// StandardPLC/Application/SaveEngine/SaveEngineMode_10
PROGRAM SaveEngineMode_10
VAR
(*	DonglitouBlink:BLINK;//0
	DonglitouBlink_biaozhi:BOOL;//0
	DOH_Y50_1: BOOL;//0
	Rotation_late:TOF;//0
	PWM_Y23_SET_Taget: UINT;//0
	PWM_Y24_SET_Taget: UINT;//0
	PWM_Y61_SET_Tatget: UINT;//0
	PWM_Y12_SET_Tatget: UINT;//0
	PWM_Y14_SET_Tatget: UINT;//0
	PWM_Y60_SET_Tatget: UINT;//0
	PWM_Y11_SET_Tatget: UINT;//0
	PWM_Y13_SET_Tatget: UINT;//0
	PWM_Y61_SET_Tatget1: INT;//0
	PWM_Y12_SET_Tatget1: INT;//0
	PWM_Y14_SET_Tatget1: INT;//0
	PWM_Y60_SET_Tatget1: INT;//0
	PWM_Y11_SET_Tatget1: INT;//0
	PWM_Y13_SET_Tatget1: INT;//0
	TIME_200ms:TON;//0
	TIME_400ms:TON;//0
	CANI_JOYX_R_last:UINT;//0
	Sub_Joyx_r: INT;//0
	curve1:curve_quxian;//0
	curve2:curve_quxian;//0
	curve3:curve_quxian;//0
	curve4:curve_quxian;//0
	curve5:curve_quxian;//0
	curve6:curve_quxian;//0
	RAMP1:RAMP_INT;//0
	RAMP2:RAMP_INT;//0
	RAMP3:RAMP_INT;//0
	RAMP4:RAMP_INT;//0
	RAMP5:RAMP_INT;//0
	RAMP6:RAMP_INT;//0
	F_RAMP_1:INT:=250;//0
	PWM_JOYX_R_UP_a:UINT;//0
	PWM_JOYX_R_UP_b:UINT;//0
	
	PWM_JOYX_R_DOWN_a:UINT;//0
	PWM_JOYX_R_DOWN_b:UINT;//0
	
	PWM_JOYY_L_DOWN_a:UINT;//0
	PWM_JOYY_L_DOWN_b:UINT;//0
	
	PWM_JOYY_L_UP_a:UINT;//0
	PWM_JOYY_L_UP_b:UINT;//0
	JOY_PAOTU:BOOL;//0
	TIME_1000_1ms:ton;//0
	tempbool:BOOL;//0
	Rtrig_d1:R_TRIG;//0
	Rtrig_d2:R_TRIG;//0
*)
END_VAR


(*******************节能控制阀主阀主泵输出执行**************************)
	
//ELSIF(GVL_SaveEngine.SaveEngineMode=10)THEN  //下放能量过高模式,先按常规执行
	//GVL_SaveEngine.Y72OutPutState:=0;
	//GVL_SaveEngine.Y71OutPutState:=0;
	GVL_SaveEngine.Y72OutPutState:=0;
	IF Mode10Timer>0 THEN
		GVL_SaveEngine.Y71OutPutState:=0;
	END_IF
	
	DOH_Y56:=FALSE;
	Y73:=FALSE;	
	PWM_Y1_Target:=REAL_TO_UINT(UINT_TO_REAL(PWM_JOYY_L_UP)/1000*(PAR_Y1_PosFull-PAR_Y1_NegFull)+PAR_Y1_NegFull);
	PWM_Y2_Target:=REAL_TO_UINT(UINT_TO_REAL(PWM_JOYY_L_UP)/1000*(PAR_Y2_PosFull-PAR_Y2_NegFull)+PAR_Y2_NegFull);
	PWM_Y8_SET_Target:=REAL_TO_UINT(UINT_TO_REAL(PWM_JOYY_L_UP)/1000*(PAR_Valve1_PosFull-PAR_Valve1_NegFull)+PAR_Valve1_NegFull);
	PWM_Y10_SET_Target:=REAL_TO_UINT(UINT_TO_REAL(PWM_JOYY_L_UP)/1000*(PAR_Valve2_PosFull-PAR_Valve2_NegFull)+PAR_Valve2_NegFull);
	PWM_Y7_SET_Target:=0;
	PWM_Y9_SET_Target:=0;
	PWM_Y33_SET_Target:=370;
	
  //Y33输出处理
	IF PWM_Y33_SET>=PWM_Y33_SET_Target THEN
	PWM_Y33_SET := PWM_Y33_SET_Target;
	END_IF
		
	IF(PWM_Y33_SET<PWM_Y33_SET_Target) THEN
		PWM_Y33_SET:=REAL_TO_UINT(UINT_TO_REAL(PWM_Y33_SET)+JianGE6);
	END_IF
	
	IF DIL_SQ3 THEN
		PWM_Y33_SET:=0;
	END_IF
(*主泵功率控制*)

//区分发动机转速
MainPump_Pressure_Taget1450:=PAR_NegFull_x;
MainPump_Pressure_Taget1600:=PAR_PosFull_x;
MainPump_Pressure_Taget1750:=PAR_Zero_x;
IF EngineSpeedTarget<=1080 THEN SPEED_CASE:=1;
ELSIF EngineSpeedTarget>1080 AND EngineSpeedTarget<=1300 THEN SPEED_CASE:=2;
ELSIF EngineSpeedTarget>1300 AND EngineSpeedTarget<=1520 THEN SPEED_CASE:=3;
ELSIF EngineSpeedTarget>1520 AND EngineSpeedTarget<=1680 THEN SPEED_CASE:=4;
ELSIF EngineSpeedTarget>1680 AND EngineSpeedTarget<=1820 THEN SPEED_CASE:=5;
ELSIF EngineSpeedTarget>1820 THEN SPEED_CASE:=6;;END_IF
//不同转速下的发动机最大功率*)
CASE SPEED_CASE OF
1:  Enginer_Power:=135;
2:  Enginer_Power:=174;
3:  Enginer_Power:=200;
4:  Enginer_Power:=230;
5:  Enginer_Power:=250;
6:  Enginer_Power:=261;
END_CASE
//不同转速下的压力值
IF(CANO_Fubeng_Press>100)THEN
	CASE SPEED_CASE OF
	1:MainPump_Pressure_Taget:=MainPump_Pressure_Taget1000-HELIU_Press_Target1000;
	2:MainPump_Pressure_Taget:=MainPump_Pressure_Taget1200-HELIU_Press_Target1200;
	3:MainPump_Pressure_Taget:=MainPump_Pressure_Taget1450-HELIU_Press_Target1400;
	4:MainPump_Pressure_Taget:=MainPump_Pressure_Taget1600-HELIU_Press_Target1600;
	5:MainPump_Pressure_Taget:=MainPump_Pressure_Taget1750-HELIU_Press_Target1800;
	6:MainPump_Pressure_Taget:=MainPump_Pressure_Taget1900-HELIU_Press_Target1900;
	END_CASE
ELSE
	CASE SPEED_CASE OF
	1:MainPump_Pressure_Taget:=MainPump_Pressure_Taget1000;
	2:MainPump_Pressure_Taget:=MainPump_Pressure_Taget1200;
	3:MainPump_Pressure_Taget:=MainPump_Pressure_Taget1450;
	4:MainPump_Pressure_Taget:=MainPump_Pressure_Taget1600;
	5:MainPump_Pressure_Taget:=MainPump_Pressure_Taget1750;
	6:MainPump_Pressure_Taget:=MainPump_Pressure_Taget1900;
	END_CASE		
END_IF

IF( CANI_ECOSwitch) THEN
	CASE SPEED_CASE OF
	1:MainPump_Pressure_Taget:=MainPump_Pressure_Taget1000-ECO_Press_Target1000;
	2:MainPump_Pressure_Taget:=MainPump_Pressure_Taget1200-ECO_Press_Target1200;
	3:MainPump_Pressure_Taget:=MainPump_Pressure_Taget1450-ECO_Press_Target1400;
	4:MainPump_Pressure_Taget:=MainPump_Pressure_Taget1600-ECO_Press_Target1600;
	5:MainPump_Pressure_Taget:=MainPump_Pressure_Taget1750-ECO_Press_Target1800;
	6:MainPump_Pressure_Taget:=MainPump_Pressure_Taget1900-ECO_Press_Target1900;
	END_CASE
END_IF
MainPump_Pressure:=CANO_MainPUMP_Press1+CANO_MainPUMP_Press2;
//消除滤波
MainPump_Pressure_Subtract:= UINT_TO_INT(MainPump_Pressure-MainPump_Pressure_last1);


//大范围波动
IF MainPump_Pressure_Subtract>270 OR MainPump_Pressure_Subtract<-270 THEN
	Subtract:=TRUE;
ELSE
	Subtract:=FALSE;	
END_IF
	TIME_LvBo4(IN:=Subtract,PT:=T#10MS);
	
IF(TIME_LvBo4.Q) AND (CANO_MainPUMP_Press1>210) THEN 
		MainPump_Pressure_ChangeBool1:=TRUE;
END_IF
	TIME_LvBo1(IN:=MainPump_Pressure_ChangeBool1,PT:=T#2S);
IF(TIME_LvBo1.Q) THEN
	MainPump_Pressure_ChangeBool1 :=FALSE;
END_IF

IF(MainPump_Pressure_ChangeBool1) AND (MainPump_Pressure>MainPump_Pressure_last1) THEN 
	MainPump_Pressure_last1:=MainPump_Pressure;
END_IF

//小范围波动
t_powertime:=TO_TIME(PAR_DeadBand_x);
IF (NOT MainPump_Pressure_ChangeBool1) THEN
	IF(MainPump_Pressure_Subtract>40 OR MainPump_Pressure_Subtract<-40)THEN 
		MainPump_Pressure_ChangeBool:=TRUE;
	ELSE
		MainPump_Pressure_ChangeBool:=FALSE;
	END_IF

	TIME_LvBo2(IN:=MainPump_Pressure_ChangeBool,PT:=t_powertime);
	IF(TIME_LvBo2.Q )THEN
		MainPump_Pressure_last1:=MainPump_Pressure;
	END_IF	
END_IF


IF PowerHead_move AND NOT(MainWinch_move) THEN
		JianGE2:=0.005;
ELSE
	IF(EngineSpeedTarget>1000 AND EngineSpeedTarget<1300)THEN
		JianGE2:=0.005;
	ELSE
		JianGE2:=0.005;
	END_IF
END_IF

IF MainPump_Pressure_last1>MainPump_Pressure_Taget THEN
	Pressure_Coe_Taget:=UINT_TO_REAL(MainPump_Pressure_Taget)/UINT_TO_REAL(MainPump_Pressure_last1);(*压力系数*)
ELSE
	Pressure_Coe_Taget:=1;
END_IF
Pressure_Coe := Pressure_Coe_Taget;


IF MainPump_Pressure_last1>MainPump_Pressure_Taget  THEN
	IF(PWM_Y1_Target>=PAR_Y1_1_NegFull)THEN
		PWM_Y1_Target_OutPut:=REAL_TO_UINT(UINT_TO_REAL(PWM_Y1_Target-PAR_Y1_1_NegFull)*Pressure_Coe+PAR_Y1_1_NegFull);
	END_IF
	IF(PWM_Y2_Target>=PAR_Y1_1_NegFull)THEN
		PWM_Y2_Target_OutPut:=REAL_TO_UINT(UINT_TO_REAL(PWM_Y2_Target-PAR_Y1_1_NegFull)*Pressure_Coe+PAR_Y1_1_NegFull);
	END_IF
ELSE
	PWM_Y1_Target_OutPut:=PWM_Y1_Target;
	PWM_Y2_Target_OutPut:=PWM_Y2_Target;
END_IF

//PWM_Y1_Target_OutPut:=PWM_Y1_Target;
//PWM_Y2_Target_OutPut:=PWM_Y2_Target;


IF(EngineSpeedTarget>CANO_SPEED AND CANO_SPEED>400)THEN
	EngineSpeedSub:=EngineSpeedTarget - CANO_SPEED;
ELSE
	EngineSpeedSub:=0;
END_IF

IF(PWM_Y1_Target_OutPut<300)THEN PWM_Y1_Target_OutPut:=300;END_IF	
IF(PWM_Y2_Target_OutPut<300)THEN PWM_Y2_Target_OutPut:=300;END_IF

RAMP15_IN:=PWM_Y1_Target_OutPut;
RAMP16_IN:=PWM_Y2_Target_OutPut;
(*
RAMP15(
	IN:=UINT_TO_INT(RAMP15_IN), 
	ASCEND:= 300, 
	DESCEND:= 400, 
	TIMEBASE:=T#1000MS , 
	RESET:=FALSE , 
	OUT=>(PWM_Y1_SET));
	
RAMP16(
	IN:=UINT_TO_INT(RAMP16_IN), 
	ASCEND:= 300, 
	DESCEND:= 400, 
	TIMEBASE:=T#1000MS , 
	RESET:=FALSE , 
	OUT=>(PWM_Y2_SET));
	*)
	
	CASE SPEED_CASE OF
                1:F_RAMP_pump:=1500; R_RAMP_pump:=100;                  
                2: 		IF MainWinch_move AND (JiaYa_move OR CANO_JiayaPressure>80)  THEN    //3泵同时起压时，降低主泵的加载速度，避免掉速熄火
                                F_RAMP_pump:=1500; R_RAMP_pump:=100;
                        ELSE
                                F_RAMP_pump:=1500; R_RAMP_pump:=100;//从200降
                                IF  PWM_JOYY_L_UP>10 THEN
                                 F_RAMP_pump:=1500; R_RAMP_pump:=200;
                                END_IF
                        END_IF            
                3:
                        IF MainWinch_move AND (JiaYa_move OR CANO_JiayaPressure>80)  THEN    //3泵同时起压时，降低主泵的加载速度，避免掉速熄火
                                F_RAMP_pump:=1500; R_RAMP_pump:=150;
                        ELSE
                                F_RAMP_pump:=1500; R_RAMP_pump:=TO_INT(PAR_NegFull_y);
                                IF  PWM_JOYY_L_UP>10 THEN
                                 F_RAMP_pump:=1500; R_RAMP_pump:=300;
                                END_IF
                        END_IF                
                4:
                        IF MainWinch_move AND (JiaYa_move OR CANO_JiayaPressure>80)  THEN
                                F_RAMP_pump:=1500; R_RAMP_pump:=150;
                        ELSE
                                F_RAMP_pump:=1500; R_RAMP_pump:=TO_INT(PAR_PosFull_y);//从200降
                                IF  PWM_JOYY_L_UP>10 THEN
                                 F_RAMP_pump:=1500; R_RAMP_pump:=300;
                                END_IF
                        END_IF                                
                5:
                        IF MainWinch_move AND (JiaYa_move OR CANO_JiayaPressure>80)  THEN
                                F_RAMP_pump:=1500; R_RAMP_pump:=200;
                        ELSE
                                F_RAMP_pump:=1500; R_RAMP_pump:=TO_INT(PAR_Zero_y);
                                IF  PWM_JOYY_L_UP>10 THEN
                                 F_RAMP_pump:=1500; R_RAMP_pump:=300;
                                END_IF
                        END_IF                        
                6:		IF MainWinch_move AND (JiaYa_move OR CANO_JiayaPressure>80)  THEN
                                F_RAMP_pump:=1500; R_RAMP_pump:=200;
                        ELSE
                                F_RAMP_pump:=1500; R_RAMP_pump:=200;
                                IF  PWM_JOYY_L_UP>10 THEN
                                 F_RAMP_pump:=1500; R_RAMP_pump:=300;
                                END_IF
                        END_IF  	
	END_CASE	
(******斜坡增步长300 斜坡降步长300->400*****)	
RAMP15(
	IN:=UINT_TO_INT(RAMP15_IN), 
	ASCEND:= R_RAMP_pump, 
	DESCEND:= 1500, 
	TIMEBASE:=T#1000MS , 
	RESET:=FALSE , 
	OUT=>(PWM_Y1_SET));
(******减斜坡300->400*****)	
RAMP16(
	IN:=UINT_TO_INT(RAMP16_IN), 
	ASCEND:= R_RAMP_pump, 
	DESCEND:= 1500, 
	TIMEBASE:=T#1000MS , 
	RESET:=FALSE , 
	OUT=>(PWM_Y2_SET));

(*
IF MainWinch_move  OR  LeftMove_move OR RightMove_move THEN  
	TIMEBASE_pump:=T#1000MS;
	TIMEBASE_xiehe:=T#500MS;
ELSE
	TIMEBASE_pump:=T#400MS;
	TIMEBASE_xiehe:=T#200MS;
END_IF
t_PowerHead_move(IN:= MainWinch_move,PT:=T#2S);
IF t_PowerHead_move.Q THEN
	F_RAMP_pump:=x_t_PowerHead_move;
	R_RAMP_pump:=x2_t_PowerHead_move;
ELSE
	F_RAMP_pump:=1000;
	R_RAMP_pump:=300;
END_IF
*)
(*
RAMP15(
	IN:=UINT_TO_INT(RAMP15_IN), 
	ASCEND:= R_RAMP_pump, 
	DESCEND:= F_RAMP_pump, 
	TIMEBASE:=TIMEBASE_pump , 
	RESET:=FALSE , 
	OUT=>(PWM_Y1_SET));
	
RAMP16(
	IN:=UINT_TO_INT(RAMP16_IN), 
	ASCEND:= R_RAMP_pump, 
	DESCEND:= F_RAMP_pump, 
	TIMEBASE:=TIMEBASE_pump , 
	RESET:=FALSE , 
	OUT=>(PWM_Y2_SET));
*)


IF (NOT Rotation_move) AND (NOT MainWinch_move) AND (NOT PowerHead_move)
		AND (NOT JiaYa_move) AND (NOT ViceWinch_move)
		AND (NOT LeftMove_move) AND (NOT RightMove_move)  THEN
	PWM_Y1_Target:=0;
	PWM_Y2_Target:=0;
END_IF


IF PWM_Y1_SET<TO_INT(PAR_Y1_1_NegFull )THEN
	PWM_Y1_SET:=TO_INT(PAR_Y1_1_NegFull);
END_IF

IF PWM_Y2_SET<TO_INT(PAR_Y1_1_NegFull )THEN
	PWM_Y2_SET:=TO_INT(PAR_Y1_1_NegFull);
END_IF

IF(PWM_Y1_SET>1000) THEN
	PWM_Y1_SET := 300;
END_IF

IF(PWM_Y2_SET>1000) THEN
	PWM_Y2_SET := 300;
END_IF	
  //Y7 8 9 10处理	
		IF(PWM_Y8_SET<1000  AND  PWM_Y8_SET>=900)THEN    //主卷下放斜坡值
				F_RAMP_mainwinch_down:=200;
			
			ELSIF(PWM_Y8_SET<900)THEN
				F_RAMP_mainwinch_down:=400;
			ELSE
				F_RAMP_mainwinch_down:=400;
			END_IF
			
		IF(PWM_Y7_SET<1000  AND  PWM_Y7_SET>=900)THEN  //主卷上提斜坡值
				F_RAMP_mainwinch_down:=300;
		ELSIF(PWM_Y7_SET<900  )THEN
				F_RAMP_mainwinch_down:=200;
		ELSE
				F_RAMP_mainwinch_down:=400;
		END_IF
			
	RAMP7(
		IN:=WORD_TO_INT(PWM_Y7_SET_Target), 
		ASCEND:= R_RAMP_mainwinch, 
		DESCEND:= F_RAMP_mainwinch_up, 
		TIMEBASE:=TIMEBASE_mainwinch , 
		RESET:=FALSE , 
		OUT=>(PWM_Y7_SET_Target1));
	IF(PWM_Y7_SET_Target1>=400) THEN
		Curve_input:=TO_UINT(PWM_Y7_SET_Target1 - 400);
		IF(Curve_input>900) THEN
			Curve_input:=900;
		END_IF
		curve7(input:=REAL_TO_UINT(UINT_TO_REAL(Curve_input)*72.8),Zero:=FALSE,Full:=FALSE,
			   PAR_Progression:=Curve_Par,OutputEnable:=TRUE);
		PWM_Y7_SET:=PAR_Valve1_NegFull + REAL_TO_UINT(UINT_TO_REAL(curve7.Output)/72.8);
	ELSE
		PWM_Y7_SET:=0;
	END_IF
	
	
	RAMP8(
		IN:=WORD_TO_INT(PWM_Y8_SET_Target), 
		ASCEND:= R_RAMP_mainwinch, 
		DESCEND:= F_RAMP_mainwinch_down, 
		TIMEBASE:=TIMEBASE_mainwinch , 
		RESET:=FALSE , 
		OUT=>(PWM_Y8_SET_Target1));
	IF(PWM_Y8_SET_Target1>=400) THEN
		Curve_input:=TO_UINT(PWM_Y8_SET_Target1 - 400);
		IF(Curve_input>900) THEN
			Curve_input:=900;
		END_IF
		curve8(input:=REAL_TO_UINT(UINT_TO_REAL(Curve_input)*72.8),Zero:=FALSE,Full:=FALSE,
			   PAR_Progression:=Curve_Par,OutputEnable:=TRUE);
		PWM_Y8_SET:=PAR_Valve1_NegFull + REAL_TO_UINT(UINT_TO_REAL(curve8.Output)/72.8);
	ELSE
		PWM_Y8_SET:=0;
	END_IF
	
	
	RAMP9(
		IN:=WORD_TO_INT(PWM_Y9_SET_Target), 
		ASCEND:= R_RAMP_mainwinch, 
		DESCEND:= F_RAMP_mainwinch_up, 
		TIMEBASE:=TIMEBASE_mainwinch , 
		RESET:=FALSE , 
		OUT=>(PWM_Y9_SET_Target1));
	IF(PWM_Y9_SET_Target1>=400) THEN
		Curve_input:=TO_UINT(PWM_Y9_SET_Target1 - 400);
		IF(Curve_input>900) THEN
			Curve_input:=900;
		END_IF
		curve9(input:=REAL_TO_UINT(UINT_TO_REAL(Curve_input)*72.8),Zero:=FALSE,Full:=FALSE,
			   PAR_Progression:=Curve_Par,OutputEnable:=TRUE);
		PWM_Y9_SET:=PAR_Valve1_NegFull + REAL_TO_UINT(UINT_TO_REAL(curve9.Output)/72.8);
	ELSE
		PWM_Y9_SET:=0;
	END_IF
	
	RAMP10(
		IN:=WORD_TO_INT(PWM_Y10_SET_Target), 
		ASCEND:= R_RAMP_mainwinch, 
		DESCEND:= F_RAMP_mainwinch_down, 
		TIMEBASE:=TIMEBASE_mainwinch , 
		RESET:=FALSE , 
		OUT=>(PWM_Y10_SET_Target1));
	IF(PWM_Y10_SET_Target1>=400) THEN
		Curve_input:=TO_UINT(PWM_Y10_SET_Target1 - 400);
		IF(Curve_input>900) THEN
			Curve_input:=900;
		END_IF
		curve10(input:=REAL_TO_UINT(UINT_TO_REAL(Curve_input)*72.8),Zero:=FALSE,Full:=FALSE,
			   PAR_Progression:=Curve_Par,OutputEnable:=TRUE);
		PWM_Y10_SET:=PAR_Valve1_NegFull + REAL_TO_UINT(UINT_TO_REAL(curve10.Output)/72.8);
	ELSE
		PWM_Y10_SET:=0;
	END_IF
    //Y7 8 9 10范围限制
	IF(PWM_Y7_SET>1300)THEN
		PWM_Y7_SET :=1300;
	END_IF
	IF(PWM_Y8_SET>1300)THEN
		PWM_Y8_SET :=1300;
	END_IF
	IF(PWM_Y9_SET>1300)THEN
		PWM_Y9_SET :=1300;
	END_IF
	IF(PWM_Y10_SET>1300)THEN
		PWM_Y10_SET :=1300;
	END_IF
	
	IF(PWM_Y7_SET<=300)THEN
		PWM_Y7_SET :=0;
	END_IF
	IF(PWM_Y8_SET<=300)THEN
		PWM_Y8_SET :=0;
	END_IF
	IF(PWM_Y9_SET<=300)THEN
		PWM_Y9_SET :=0;
	END_IF
	IF(PWM_Y10_SET<=300)THEN
		PWM_Y10_SET :=0;
	END_IF
	(*主泵卸荷阀控制*)
		PWM_Y39_SET_Target:=MAX(PWM_Y8_SET_Target,PWM_Y7_SET_Target);
		PWM_Y40_SET_Target:=MAX(PWM_Y9_SET_Target,PWM_Y10_SET_Target);
	(*卸荷动作缓冲*)
RAMP19(
	IN:=WORD_TO_INT(PWM_Y39_SET_Target), 
	ASCEND:= R_RAMP_xiehe, 
	DESCEND:= F_RAMP_xiehe, 
	TIMEBASE:=TIMEBASE_xiehe , 
	RESET:=FALSE , 
	OUT=>(PWM_Y39_SET_Target1));
IF(PWM_Y39_SET_Target1>=400) THEN
	Curve_input:=TO_UINT(PWM_Y39_SET_Target1 - 400);
	IF(Curve_input>900) THEN
		Curve_input:=900;
	END_IF
	curve19(input:=REAL_TO_UINT(UINT_TO_REAL(Curve_input)*72.8),Zero:=FALSE,Full:=FALSE,
		   PAR_Progression:=Curve_Par1,OutputEnable:=TRUE);
	PWM_Y39_SET:=PAR_Valve1_NegFull + REAL_TO_UINT(UINT_TO_REAL(curve19.Output)/72.8);
ELSE
	PWM_Y39_SET:=0;
END_IF


RAMP20(
	IN:=WORD_TO_INT(PWM_Y40_SET_Target), 
	ASCEND:= R_RAMP_xiehe, 
	DESCEND:= F_RAMP_xiehe, 
	TIMEBASE:=TIMEBASE_xiehe , 
	RESET:=FALSE , 
	OUT=>(PWM_Y40_SET_Target1));
IF(PWM_Y40_SET_Target1>=400) THEN
	Curve_input:=TO_UINT(PWM_Y40_SET_Target1 - 400);
	IF(Curve_input>900) THEN
		Curve_input:=900;
	END_IF
	curve20(input:=REAL_TO_UINT(UINT_TO_REAL(Curve_input)*72.8),Zero:=FALSE,Full:=FALSE,
		   PAR_Progression:=Curve_Par1,OutputEnable:=TRUE);
	PWM_Y40_SET:=PAR_Valve1_NegFull + REAL_TO_UINT(UINT_TO_REAL(curve20.Output)/72.8);
ELSE
	PWM_Y40_SET:=0;
END_IF
	
IF(PWM_Y39_SET>1300)THEN
	PWM_Y39_SET :=1300;
END_IF
IF(PWM_Y40_SET>1300)THEN
	PWM_Y40_SET :=1300;
END_IF

IF(PWM_Y39_SET<=300)THEN
	PWM_Y39_SET :=0;
END_IF
IF(PWM_Y40_SET<=300)THEN
	PWM_Y40_SET :=0;
END_IF

END_PROGRAM

// StandardPLC/Application/SaveEngine/SaveEngineMode_11
PROGRAM SaveEngineMode_11
VAR

	TON1: TON;
	TON2: TON;
	AI_PM2Pre_Flag1: BOOL;
	AI_PM2Pre_Flag3: BOOL;
	PM2Pre_Rtrig1: R_TRIG;
	PM2Pre_Rtrig3: R_TRIG;
	Mod1CasePWM_Y1: UINT;
END_VAR

(*******************节能控制阀主阀主泵输出执行**************************)
	
//ELSIF(GVL_SaveEngine.SaveEngineMode=11)THEN  //下放入口压力过高模式,
	

	//GVL_SaveEngine.Y72OutPutState:=0;
	//GVL_SaveEngine.Y71OutPutState:=0;
	(****先关Y72 再关Y71间隔100ms****)
	GVL_SaveEngine.Y72OutPutState:=0;
	IF Mode11Timer>0 THEN
		GVL_SaveEngine.Y71OutPutState:=0;
	END_IF
	
	DOH_Y56:=FALSE;
	Y73:=FALSE;	
	//PWM_Y1_Target:=REAL_TO_UINT(UINT_TO_REAL(PWM_JOYY_L_UP)/1000*(PAR_Y1_PosFull-PAR_Y1_NegFull)+PAR_Y1_NegFull);
	//PWM_Y2_Target:=REAL_TO_UINT(UINT_TO_REAL(PWM_JOYY_L_UP)/1000*(PAR_Y2_PosFull-PAR_Y2_NegFull)+PAR_Y2_NegFull);
	//PWM_Y8_SET_Target:=REAL_TO_UINT(UINT_TO_REAL(PWM_JOYY_L_UP)/1000*(PAR_Valve1_PosFull-PAR_Valve1_NegFull)+PAR_Valve1_NegFull);
	//PWM_Y10_SET_Target:=REAL_TO_UINT(UINT_TO_REAL(PWM_JOYY_L_UP)/1000*(PAR_Valve2_PosFull-PAR_Valve2_NegFull)+PAR_Valve2_NegFull);
	//PWM_Y7_SET_Target:=0;
	//PWM_Y9_SET_Target:=0;
	//PWM_Y33_SET_Target:=370;
  //Y33输出处理
  
  	TON1(IN:=NOT TON1.Q AND GVL_SaveEngine.AI_PM2Pre<30 ,PT:=T#200MS);
	TON2(IN:=NOT TON2.Q AND GVL_SaveEngine.AI_PM2Pre>=60 ,PT:=T#1S);
	IF TON2.Q AND GVL_SaveEngine.PWM_Y33_SET_Target<500 THEN
		AI_PM2Pre_Flag1:=TRUE;
	ELSE
		AI_PM2Pre_Flag1:=FALSE;
	END_IF
	IF GVL_SaveEngine.PWM_Y33_SET_Target>=230 AND TON1.Q  THEN
		AI_PM2Pre_Flag3:=TRUE;
	ELSE
		AI_PM2Pre_Flag3:=FALSE;
	END_IF

	PM2Pre_Rtrig1(CLK:=AI_PM2Pre_Flag1);
	PM2Pre_Rtrig3(CLK:=AI_PM2Pre_Flag3);

	IF(PM2Pre_Rtrig1.Q)THEN
		//A:=A+1;
		GVL_SaveEngine.PWM_Y33_SET_Target:=GVL_SaveEngine.PWM_Y33_SET_Target+17;
		AI_PM2Pre_Flag1:=FALSE;
	END_IF
	
	IF(PM2Pre_Rtrig3.Q)THEN
		//B:=B+1;
		GVL_SaveEngine.PWM_Y33_SET_Target:=GVL_SaveEngine.PWM_Y33_SET_Target-17;
		AI_PM2Pre_Flag3:=FALSE;
	END_IF
	GVL_SaveEngine.PWM_Y33_SET_Target:=LIMIT(417,GVL_SaveEngine.PWM_Y33_SET_Target,465);
	PWM_Y33_SET := GVL_SaveEngine.PWM_Y33_SET_Target;//去掉原有坡度执行防止干扰
	
	(*IF PWM_Y33_SET>=PWM_Y33_SET_Target THEN
	PWM_Y33_SET := PWM_Y33_SET_Target;
	END_IF
		
	IF(PWM_Y33_SET<PWM_Y33_SET_Target) THEN
		PWM_Y33_SET:=REAL_TO_UINT(UINT_TO_REAL(PWM_Y33_SET)+JianGE6);
	END_IF
	*)
	IF DIL_SQ3 THEN
		PWM_Y33_SET:=0;
	END_IF
	//和1模式一样，根据档位设定目标电流，以及主卷排量计算主泵最大电流
	CASE AI_ECM2_Flag OF
			1: Mod1CasePWM_Y1:=REAL_TO_UINT(362.5+47.8*30/1100*(600-PWM_Y33_SET)/1.85)+40;
			2: Mod1CasePWM_Y1:=REAL_TO_UINT(362.5+47.8*42/1200*(600-PWM_Y33_SET)/1.85)+40;
			3: Mod1CasePWM_Y1:=REAL_TO_UINT(362.5+47.8*55/1450*(600-PWM_Y33_SET)/1.85)+40;
			4: Mod1CasePWM_Y1:=REAL_TO_UINT(362.5+47.8*62/1500*(600-PWM_Y33_SET)/1.85)+120;//调速 55-100
			5: Mod1CasePWM_Y1:=REAL_TO_UINT(362.5+47.8*68/1500*(600-PWM_Y33_SET)/1.85)+120;//0-75
			6: Mod1CasePWM_Y1:=REAL_TO_UINT(362.5+47.8*72/1500*(600-PWM_Y33_SET)/1.85)+120;//-20-75
	END_CASE
		
	(****前400ms 11模式输出电流给大****)		
	(*IF Mode11Timer<4 THEN
		CASE AI_ECM2_Flag OF
			1: Mod1CasePWM_Y1:=REAL_TO_UINT(362.5+47.8*30/1100*(600-PWM_Y33_SET)/1.85)+40;
			2: Mod1CasePWM_Y1:=REAL_TO_UINT(362.5+47.8*42/1200*(600-PWM_Y33_SET)/1.85)+40;
			3: Mod1CasePWM_Y1:=REAL_TO_UINT(362.5+47.8*55/1450*(600-PWM_Y33_SET)/1.85)+40;
			4: Mod1CasePWM_Y1:=REAL_TO_UINT(362.5+47.8*62/1500*(600-PWM_Y33_SET)/1.85)+80;//调速
			5: Mod1CasePWM_Y1:=REAL_TO_UINT(362.5+47.8*68/1500*(600-PWM_Y33_SET)/1.85)+0;//
			6: Mod1CasePWM_Y1:=REAL_TO_UINT(362.5+47.8*72/1500*(600-PWM_Y33_SET)/1.85)-20;//
		END_CASE
	END_IF
	*)
		
	PWM_Y1_Target:=REAL_TO_UINT(UINT_TO_REAL(PWM_JOYY_L_UP)/1000*(Mod1CasePWM_Y1-PAR_Y1_NegFull)+PAR_Y1_NegFull);
	PWM_Y2_Target:=REAL_TO_UINT(UINT_TO_REAL(PWM_JOYY_L_UP)/1000*(Mod1CasePWM_Y1-PAR_Y2_NegFull)+PAR_Y2_NegFull);
	IF PWM_Y1_Target>700 THEN 
		PWM_Y1_Target:=700;
	END_IF
	IF PWM_Y2_Target>700 THEN 
		PWM_Y2_Target:=700;
	END_IF
	
	//PWM_Y1_SET:=UINT_TO_INT(PWM_Y1_Target);
	//PWM_Y2_SET:=UINT_TO_INT(PWM_Y2_Target); 3.15未注释
	 
	
(*主泵功率控制*)

//区分发动机转速
MainPump_Pressure_Taget1450:=PAR_NegFull_x;
MainPump_Pressure_Taget1600:=PAR_PosFull_x;
MainPump_Pressure_Taget1750:=PAR_Zero_x;
IF EngineSpeedTarget<=1080 THEN SPEED_CASE:=1;
ELSIF EngineSpeedTarget>1080 AND EngineSpeedTarget<=1300 THEN SPEED_CASE:=2;
ELSIF EngineSpeedTarget>1300 AND EngineSpeedTarget<=1520 THEN SPEED_CASE:=3;
ELSIF EngineSpeedTarget>1520 AND EngineSpeedTarget<=1680 THEN SPEED_CASE:=4;
ELSIF EngineSpeedTarget>1680 AND EngineSpeedTarget<=1820 THEN SPEED_CASE:=5;
ELSIF EngineSpeedTarget>1820 THEN SPEED_CASE:=6;;END_IF
//不同转速下的发动机最大功率*)
CASE SPEED_CASE OF
1:  Enginer_Power:=135;
2:  Enginer_Power:=174;
3:  Enginer_Power:=200;
4:  Enginer_Power:=230;
5:  Enginer_Power:=250;
6:  Enginer_Power:=261;
END_CASE
//不同转速下的压力值
IF(CANO_Fubeng_Press>100)THEN
	CASE SPEED_CASE OF
	1:MainPump_Pressure_Taget:=MainPump_Pressure_Taget1000-HELIU_Press_Target1000;
	2:MainPump_Pressure_Taget:=MainPump_Pressure_Taget1200-HELIU_Press_Target1200;
	3:MainPump_Pressure_Taget:=MainPump_Pressure_Taget1450-HELIU_Press_Target1400;
	4:MainPump_Pressure_Taget:=MainPump_Pressure_Taget1600-HELIU_Press_Target1600;
	5:MainPump_Pressure_Taget:=MainPump_Pressure_Taget1750-HELIU_Press_Target1800;
	6:MainPump_Pressure_Taget:=MainPump_Pressure_Taget1900-HELIU_Press_Target1900;
	END_CASE
ELSE
	CASE SPEED_CASE OF
	1:MainPump_Pressure_Taget:=MainPump_Pressure_Taget1000;
	2:MainPump_Pressure_Taget:=MainPump_Pressure_Taget1200;
	3:MainPump_Pressure_Taget:=MainPump_Pressure_Taget1450;
	4:MainPump_Pressure_Taget:=MainPump_Pressure_Taget1600;
	5:MainPump_Pressure_Taget:=MainPump_Pressure_Taget1750;
	6:MainPump_Pressure_Taget:=MainPump_Pressure_Taget1900;
	END_CASE		
END_IF

IF( CANI_ECOSwitch) THEN
	CASE SPEED_CASE OF
	1:MainPump_Pressure_Taget:=MainPump_Pressure_Taget1000-ECO_Press_Target1000;
	2:MainPump_Pressure_Taget:=MainPump_Pressure_Taget1200-ECO_Press_Target1200;
	3:MainPump_Pressure_Taget:=MainPump_Pressure_Taget1450-ECO_Press_Target1400;
	4:MainPump_Pressure_Taget:=MainPump_Pressure_Taget1600-ECO_Press_Target1600;
	5:MainPump_Pressure_Taget:=MainPump_Pressure_Taget1750-ECO_Press_Target1800;
	6:MainPump_Pressure_Taget:=MainPump_Pressure_Taget1900-ECO_Press_Target1900;
	END_CASE
END_IF
MainPump_Pressure:=CANO_MainPUMP_Press1+CANO_MainPUMP_Press2;
//消除滤波
MainPump_Pressure_Subtract:= UINT_TO_INT(MainPump_Pressure-MainPump_Pressure_last1);


//大范围波动
IF MainPump_Pressure_Subtract>270 OR MainPump_Pressure_Subtract<-270 THEN
	Subtract:=TRUE;
ELSE
	Subtract:=FALSE;	
END_IF
	TIME_LvBo4(IN:=Subtract,PT:=T#10MS);
	
IF(TIME_LvBo4.Q)  AND (CANO_MainPUMP_Press1>210) THEN 
		MainPump_Pressure_ChangeBool1:=TRUE;
END_IF
	TIME_LvBo1(IN:=MainPump_Pressure_ChangeBool1,PT:=T#2S);
IF(TIME_LvBo1.Q) THEN
	MainPump_Pressure_ChangeBool1 :=FALSE;
END_IF

IF(MainPump_Pressure_ChangeBool1) AND (MainPump_Pressure>MainPump_Pressure_last1) THEN 
	MainPump_Pressure_last1:=MainPump_Pressure;
END_IF

//小范围波动
t_powertime:=TO_TIME(PAR_DeadBand_x);
IF (NOT MainPump_Pressure_ChangeBool1) THEN
	IF(MainPump_Pressure_Subtract>40 OR MainPump_Pressure_Subtract<-40)THEN 
		MainPump_Pressure_ChangeBool:=TRUE;
	ELSE
		MainPump_Pressure_ChangeBool:=FALSE;
	END_IF

	TIME_LvBo2(IN:=MainPump_Pressure_ChangeBool,PT:=t_powertime);
	IF(TIME_LvBo2.Q )THEN
		MainPump_Pressure_last1:=MainPump_Pressure;
	END_IF	
END_IF


IF PowerHead_move AND NOT(MainWinch_move) THEN
		JianGE2:=0.005;
ELSE
	IF(EngineSpeedTarget>1000 AND EngineSpeedTarget<1300)THEN
		JianGE2:=0.005;
	ELSE
		JianGE2:=0.005;
	END_IF
END_IF

IF MainPump_Pressure_last1>MainPump_Pressure_Taget THEN
	Pressure_Coe_Taget:=UINT_TO_REAL(MainPump_Pressure_Taget)/UINT_TO_REAL(MainPump_Pressure_last1);(*压力系数*)
ELSE
	Pressure_Coe_Taget:=1;
END_IF
Pressure_Coe := Pressure_Coe_Taget;


IF MainPump_Pressure_last1>MainPump_Pressure_Taget  THEN
	IF(PWM_Y1_Target>=PAR_Y1_1_NegFull)THEN
		PWM_Y1_Target_OutPut:=REAL_TO_UINT(UINT_TO_REAL(PWM_Y1_Target-PAR_Y1_1_NegFull)*Pressure_Coe+PAR_Y1_1_NegFull);
	END_IF
	IF(PWM_Y2_Target>=PAR_Y1_1_NegFull)THEN
		PWM_Y2_Target_OutPut:=REAL_TO_UINT(UINT_TO_REAL(PWM_Y2_Target-PAR_Y1_1_NegFull)*Pressure_Coe+PAR_Y1_1_NegFull);
	END_IF
ELSE
	PWM_Y1_Target_OutPut:=PWM_Y1_Target;
	PWM_Y2_Target_OutPut:=PWM_Y2_Target;
END_IF



//PWM_Y1_Target_OutPut:=PWM_Y1_Target;
//PWM_Y2_Target_OutPut:=PWM_Y2_Target;


IF(EngineSpeedTarget>CANO_SPEED AND CANO_SPEED>400)THEN
	EngineSpeedSub:=EngineSpeedTarget - CANO_SPEED;
ELSE
	EngineSpeedSub:=0;
END_IF

IF(PWM_Y1_Target_OutPut<300)THEN PWM_Y1_Target_OutPut:=300;END_IF	
IF(PWM_Y2_Target_OutPut<300)THEN PWM_Y2_Target_OutPut:=300;END_IF

RAMP15_IN:=PWM_Y1_Target_OutPut;
RAMP16_IN:=PWM_Y2_Target_OutPut;
(*
RAMP15(
	IN:=UINT_TO_INT(RAMP15_IN), 
	ASCEND:= 300, 
	DESCEND:= 400, 
	TIMEBASE:=T#1000MS , 
	RESET:=FALSE , 
	OUT=>(PWM_Y1_SET));
	
RAMP16(
	IN:=UINT_TO_INT(RAMP16_IN), 
	ASCEND:= 300, 
	DESCEND:= 400, 
	TIMEBASE:=T#1000MS , 
	RESET:=FALSE , 
	OUT=>(PWM_Y2_SET));
*)
	CASE SPEED_CASE OF
                1:F_RAMP_pump:=1500; R_RAMP_pump:=100;                  
                2: 		IF MainWinch_move AND (JiaYa_move OR CANO_JiayaPressure>80)  THEN    //3泵同时起压时，降低主泵的加载速度，避免掉速熄火
                                F_RAMP_pump:=1500; R_RAMP_pump:=100;
                        ELSE
                                F_RAMP_pump:=1500; R_RAMP_pump:=100;//从200降
                                IF  PWM_JOYY_L_UP>10 THEN
                                 F_RAMP_pump:=1500; R_RAMP_pump:=200;
                                END_IF
                        END_IF            
                3:
                        IF MainWinch_move AND (JiaYa_move OR CANO_JiayaPressure>80)  THEN    //3泵同时起压时，降低主泵的加载速度，避免掉速熄火
                                F_RAMP_pump:=1500; R_RAMP_pump:=150;
                        ELSE
                                F_RAMP_pump:=1500; R_RAMP_pump:=TO_INT(PAR_NegFull_y);
                                IF  PWM_JOYY_L_UP>10 THEN
                                 F_RAMP_pump:=1500; R_RAMP_pump:=300;
                                END_IF
                        END_IF                
                4:
                        IF MainWinch_move AND (JiaYa_move OR CANO_JiayaPressure>80)  THEN
                                F_RAMP_pump:=1500; R_RAMP_pump:=150;
                        ELSE
                                F_RAMP_pump:=1500; R_RAMP_pump:=TO_INT(PAR_PosFull_y);//从200降
                                IF  PWM_JOYY_L_UP>10 THEN
                                 F_RAMP_pump:=1500; R_RAMP_pump:=300;
                                END_IF
                        END_IF                                
                5:
                        IF MainWinch_move AND (JiaYa_move OR CANO_JiayaPressure>80)  THEN
                                F_RAMP_pump:=1500; R_RAMP_pump:=200;
                        ELSE
                                F_RAMP_pump:=1500; R_RAMP_pump:=TO_INT(PAR_Zero_y);
                                IF  PWM_JOYY_L_UP>10 THEN
                                 F_RAMP_pump:=1500; R_RAMP_pump:=300;
                                END_IF
                        END_IF                        
                6:		IF MainWinch_move AND (JiaYa_move OR CANO_JiayaPressure>80)  THEN
                                F_RAMP_pump:=1500; R_RAMP_pump:=200;
                        ELSE
                                F_RAMP_pump:=1500; R_RAMP_pump:=200;
                                IF  PWM_JOYY_L_UP>10 THEN
                                 F_RAMP_pump:=1500; R_RAMP_pump:=300;
                                END_IF
                        END_IF  	
	END_CASE
(******斜坡增步长300 斜坡降步长300->400*****)	
RAMP15(
	IN:=UINT_TO_INT(RAMP15_IN), 
	ASCEND:= R_RAMP_pump, 
	DESCEND:= 1500, 
	TIMEBASE:=T#1000MS , 
	RESET:=FALSE , 
	OUT=>(PWM_Y1_SET));
(******减斜坡300->400*****)	
RAMP16(
	IN:=UINT_TO_INT(RAMP16_IN), 
	ASCEND:= R_RAMP_pump, 
	DESCEND:= 1500, 
	TIMEBASE:=T#1000MS , 
	RESET:=FALSE , 
	OUT=>(PWM_Y2_SET));

IF (NOT Rotation_move) AND (NOT MainWinch_move) AND (NOT PowerHead_move)
		AND (NOT JiaYa_move) AND (NOT ViceWinch_move)
		AND (NOT LeftMove_move) AND (NOT RightMove_move)  THEN
	PWM_Y1_Target:=0;
	PWM_Y2_Target:=0;
END_IF


IF PWM_Y1_SET<TO_INT(PAR_Y1_1_NegFull )THEN
	PWM_Y1_SET:=TO_INT(PAR_Y1_1_NegFull);
END_IF

IF PWM_Y2_SET<TO_INT(PAR_Y1_1_NegFull )THEN
	PWM_Y2_SET:=TO_INT(PAR_Y1_1_NegFull);
END_IF

IF(PWM_Y1_SET>1000) THEN
	PWM_Y1_SET := 300;
END_IF

IF(PWM_Y2_SET>1000) THEN
	PWM_Y2_SET := 300;
END_IF	

	PWM_Y8_SET_Target:=REAL_TO_UINT(UINT_TO_REAL(PWM_JOYY_L_UP)/1000*(PAR_Valve1_PosFull-PAR_Valve1_NegFull)+PAR_Valve1_NegFull);
	PWM_Y10_SET_Target:=REAL_TO_UINT(UINT_TO_REAL(PWM_JOYY_L_UP)/1000*(PAR_Valve2_PosFull-PAR_Valve2_NegFull)+PAR_Valve2_NegFull);
	PWM_Y7_SET_Target:=0;
	PWM_Y9_SET_Target:=0;
  //Y7 8 9 10处理	
		IF(PWM_Y8_SET<1000  AND  PWM_Y8_SET>=900)THEN    //主卷下放斜坡值
				F_RAMP_mainwinch_down:=200;
			
			ELSIF(PWM_Y8_SET<900)THEN
				F_RAMP_mainwinch_down:=400;
			ELSE
				F_RAMP_mainwinch_down:=400;
			END_IF
			
		IF(PWM_Y7_SET<1000  AND  PWM_Y7_SET>=900)THEN  //主卷上提斜坡值
				F_RAMP_mainwinch_down:=300;
		ELSIF(PWM_Y7_SET<900  )THEN
				F_RAMP_mainwinch_down:=200;
		ELSE
				F_RAMP_mainwinch_down:=400;
		END_IF
			
	RAMP7(
		IN:=WORD_TO_INT(PWM_Y7_SET_Target), 
		ASCEND:= R_RAMP_mainwinch, 
		DESCEND:= F_RAMP_mainwinch_up, 
		TIMEBASE:=TIMEBASE_mainwinch , 
		RESET:=FALSE , 
		OUT=>(PWM_Y7_SET_Target1));
	IF(PWM_Y7_SET_Target1>=400) THEN
		Curve_input:=TO_UINT(PWM_Y7_SET_Target1 - 400);
		IF(Curve_input>900) THEN
			Curve_input:=900;
		END_IF
		curve7(input:=REAL_TO_UINT(UINT_TO_REAL(Curve_input)*72.8),Zero:=FALSE,Full:=FALSE,
			   PAR_Progression:=Curve_Par,OutputEnable:=TRUE);
		PWM_Y7_SET:=PAR_Valve1_NegFull + REAL_TO_UINT(UINT_TO_REAL(curve7.Output)/72.8);
	ELSE
		PWM_Y7_SET:=0;
	END_IF
	
	
	RAMP8(
		IN:=WORD_TO_INT(PWM_Y8_SET_Target), 
		ASCEND:= R_RAMP_mainwinch, 
		DESCEND:= F_RAMP_mainwinch_down, 
		TIMEBASE:=TIMEBASE_mainwinch , 
		RESET:=FALSE , 
		OUT=>(PWM_Y8_SET_Target1));
	IF(PWM_Y8_SET_Target1>=400) THEN
		Curve_input:=TO_UINT(PWM_Y8_SET_Target1 - 400);
		IF(Curve_input>900) THEN
			Curve_input:=900;
		END_IF
		curve8(input:=REAL_TO_UINT(UINT_TO_REAL(Curve_input)*72.8),Zero:=FALSE,Full:=FALSE,
			   PAR_Progression:=Curve_Par,OutputEnable:=TRUE);
		PWM_Y8_SET:=PAR_Valve1_NegFull + REAL_TO_UINT(UINT_TO_REAL(curve8.Output)/72.8);
	ELSE
		PWM_Y8_SET:=0;
	END_IF
	
	
	RAMP9(
		IN:=WORD_TO_INT(PWM_Y9_SET_Target), 
		ASCEND:= R_RAMP_mainwinch, 
		DESCEND:= F_RAMP_mainwinch_up, 
		TIMEBASE:=TIMEBASE_mainwinch , 
		RESET:=FALSE , 
		OUT=>(PWM_Y9_SET_Target1));
	IF(PWM_Y9_SET_Target1>=400) THEN
		Curve_input:=TO_UINT(PWM_Y9_SET_Target1 - 400);
		IF(Curve_input>900) THEN
			Curve_input:=900;
		END_IF
		curve9(input:=REAL_TO_UINT(UINT_TO_REAL(Curve_input)*72.8),Zero:=FALSE,Full:=FALSE,
			   PAR_Progression:=Curve_Par,OutputEnable:=TRUE);
		PWM_Y9_SET:=PAR_Valve1_NegFull + REAL_TO_UINT(UINT_TO_REAL(curve9.Output)/72.8);
	ELSE
		PWM_Y9_SET:=0;
	END_IF
	
	RAMP10(
		IN:=WORD_TO_INT(PWM_Y10_SET_Target), 
		ASCEND:= R_RAMP_mainwinch, 
		DESCEND:= F_RAMP_mainwinch_down, 
		TIMEBASE:=TIMEBASE_mainwinch , 
		RESET:=FALSE , 
		OUT=>(PWM_Y10_SET_Target1));
	IF(PWM_Y10_SET_Target1>=400) THEN
		Curve_input:=TO_UINT(PWM_Y10_SET_Target1 - 400);
		IF(Curve_input>900) THEN
			Curve_input:=900;
		END_IF
		curve10(input:=REAL_TO_UINT(UINT_TO_REAL(Curve_input)*72.8),Zero:=FALSE,Full:=FALSE,
			   PAR_Progression:=Curve_Par,OutputEnable:=TRUE);
		PWM_Y10_SET:=PAR_Valve1_NegFull + REAL_TO_UINT(UINT_TO_REAL(curve10.Output)/72.8);
	ELSE
		PWM_Y10_SET:=0;
	END_IF
    //Y7 8 9 10范围限制
	IF(PWM_Y7_SET>1300)THEN
		PWM_Y7_SET :=1300;
	END_IF
	IF(PWM_Y8_SET>1300)THEN
		PWM_Y8_SET :=1300;
	END_IF
	IF(PWM_Y9_SET>1300)THEN
		PWM_Y9_SET :=1300;
	END_IF
	IF(PWM_Y10_SET>1300)THEN
		PWM_Y10_SET :=1300;
	END_IF
	
	IF(PWM_Y7_SET<=300)THEN
		PWM_Y7_SET :=0;
	END_IF
	IF(PWM_Y8_SET<=300)THEN
		PWM_Y8_SET :=0;
	END_IF
	IF(PWM_Y9_SET<=300)THEN
		PWM_Y9_SET :=0;
	END_IF
	IF(PWM_Y10_SET<=300)THEN
		PWM_Y10_SET :=0;
	END_IF
	
	PWM_Y7_SET:=0;
	PWM_Y9_SET:=0;
	(*主泵卸荷阀控制*)
		PWM_Y39_SET_Target:=MAX(PWM_Y8_SET_Target,PWM_Y7_SET_Target);
		PWM_Y40_SET_Target:=MAX(PWM_Y9_SET_Target,PWM_Y10_SET_Target);
	(*卸荷动作缓冲*)
RAMP19(
	IN:=WORD_TO_INT(PWM_Y39_SET_Target), 
	ASCEND:= R_RAMP_xiehe, 
	DESCEND:= F_RAMP_xiehe, 
	TIMEBASE:=TIMEBASE_xiehe , 
	RESET:=FALSE , 
	OUT=>(PWM_Y39_SET_Target1));
IF(PWM_Y39_SET_Target1>=400) THEN
	Curve_input:=TO_UINT(PWM_Y39_SET_Target1 - 400);
	IF(Curve_input>900) THEN
		Curve_input:=900;
	END_IF
	curve19(input:=REAL_TO_UINT(UINT_TO_REAL(Curve_input)*72.8),Zero:=FALSE,Full:=FALSE,
		   PAR_Progression:=Curve_Par1,OutputEnable:=TRUE);
	PWM_Y39_SET:=PAR_Valve1_NegFull + REAL_TO_UINT(UINT_TO_REAL(curve19.Output)/72.8);
ELSE
	PWM_Y39_SET:=0;
END_IF


RAMP20(
	IN:=WORD_TO_INT(PWM_Y40_SET_Target), 
	ASCEND:= R_RAMP_xiehe, 
	DESCEND:= F_RAMP_xiehe, 
	TIMEBASE:=TIMEBASE_xiehe , 
	RESET:=FALSE , 
	OUT=>(PWM_Y40_SET_Target1));

IF(PWM_Y40_SET_Target1>=400) THEN
	Curve_input:=TO_UINT(PWM_Y40_SET_Target1 - 400);
	IF(Curve_input>900) THEN
		Curve_input:=900;
	END_IF
	curve20(input:=REAL_TO_UINT(UINT_TO_REAL(Curve_input)*72.8),Zero:=FALSE,Full:=FALSE,
		   PAR_Progression:=Curve_Par1,OutputEnable:=TRUE);
	PWM_Y40_SET:=PAR_Valve1_NegFull + REAL_TO_UINT(UINT_TO_REAL(curve20.Output)/72.8);
ELSE
	PWM_Y40_SET:=0;
END_IF
	
IF(PWM_Y39_SET>1300)THEN
	PWM_Y39_SET :=1300;
END_IF
IF(PWM_Y40_SET>1300)THEN
	PWM_Y40_SET :=1300;
END_IF

IF(PWM_Y39_SET<=300)THEN
	PWM_Y39_SET :=0;
END_IF
IF(PWM_Y40_SET<=300)THEN
	PWM_Y40_SET :=0;
END_IF

END_PROGRAM

// StandardPLC/Application/SaveEngine/SaveEngineMode_12
PROGRAM SaveEngineMode_12
VAR
	PAR_Y1_PosFull:UINT:=600;
END_VAR

(*******************节能控制阀主阀主泵输出执行**************************)
	
//ELSIF(GVL_SaveEngine.SaveEngineMode=12)THEN//节能下降回至中位模式,
	//GVL_SaveEngine.Y72OutPutState:=0;
	//GVL_SaveEngine.Y71OutPutState:=0;
	(****先关Y72再关Y71减少回中位时M1压力冲击****)
	GVL_SaveEngine.Y72OutPutState:=0;
	IF Mode12Timer>0 THEN
		GVL_SaveEngine.Y71OutPutState:=0;
	END_IF
	
	Y73:=TRUE;
	PWM_Y7_SET_Target:=0;
	PWM_Y9_SET_Target:=0;
	PWM_Y8_SET_Target:=0;
	PWM_Y10_SET_Target:=0;
	RAMP7(
		IN:=WORD_TO_INT(PWM_Y7_SET_Target), 
		ASCEND:= R_RAMP_mainwinch, 
		DESCEND:= F_RAMP_mainwinch_up, 
		TIMEBASE:=TIMEBASE_mainwinch , 
		RESET:=FALSE , 
		OUT=>(PWM_Y7_SET_Target1));
	IF(PWM_Y7_SET_Target1>=400) THEN
		Curve_input:=TO_UINT(PWM_Y7_SET_Target1 - 400);
		IF(Curve_input>900) THEN
			Curve_input:=900;
		END_IF
		curve7(input:=REAL_TO_UINT(UINT_TO_REAL(Curve_input)*72.8),Zero:=FALSE,Full:=FALSE,
			   PAR_Progression:=Curve_Par,OutputEnable:=TRUE);
		PWM_Y7_SET:=PAR_Valve1_NegFull + REAL_TO_UINT(UINT_TO_REAL(curve7.Output)/72.8);
	ELSE
		PWM_Y7_SET:=0;
	END_IF
	
	RAMP8(
		IN:=WORD_TO_INT(PWM_Y8_SET_Target), 
		ASCEND:= R_RAMP_mainwinch, 
		DESCEND:= F_RAMP_mainwinch_down, 
		TIMEBASE:=TIMEBASE_mainwinch , 
		RESET:=FALSE , 
		OUT=>(PWM_Y8_SET_Target1));
	IF(PWM_Y8_SET_Target1>=400) THEN
		Curve_input:=TO_UINT(PWM_Y8_SET_Target1 - 400);
		IF(Curve_input>900) THEN
			Curve_input:=900;
		END_IF
		curve8(input:=REAL_TO_UINT(UINT_TO_REAL(Curve_input)*72.8),Zero:=FALSE,Full:=FALSE,
			   PAR_Progression:=Curve_Par,OutputEnable:=TRUE);
		PWM_Y8_SET:=PAR_Valve1_NegFull + REAL_TO_UINT(UINT_TO_REAL(curve8.Output)/72.8);
	ELSE
		PWM_Y8_SET:=0;
	END_IF
		RAMP9(
		IN:=WORD_TO_INT(PWM_Y9_SET_Target), 
		ASCEND:= R_RAMP_mainwinch, 
		DESCEND:= F_RAMP_mainwinch_up, 
		TIMEBASE:=TIMEBASE_mainwinch , 
		RESET:=FALSE , 
		OUT=>(PWM_Y9_SET_Target1));
	IF(PWM_Y9_SET_Target1>=400) THEN
		Curve_input:=TO_UINT(PWM_Y9_SET_Target1 - 400);
		IF(Curve_input>900) THEN
			Curve_input:=900;
		END_IF
		curve9(input:=REAL_TO_UINT(UINT_TO_REAL(Curve_input)*72.8),Zero:=FALSE,Full:=FALSE,
			   PAR_Progression:=Curve_Par,OutputEnable:=TRUE);
		PWM_Y9_SET:=PAR_Valve1_NegFull + REAL_TO_UINT(UINT_TO_REAL(curve9.Output)/72.8);
	ELSE
		PWM_Y9_SET:=0;
	END_IF
	
	RAMP10(
		IN:=WORD_TO_INT(PWM_Y10_SET_Target), 
		ASCEND:= R_RAMP_mainwinch, 
		DESCEND:= F_RAMP_mainwinch_down, 
		TIMEBASE:=TIMEBASE_mainwinch , 
		RESET:=FALSE , 
		OUT=>(PWM_Y10_SET_Target1));
	IF(PWM_Y10_SET_Target1>=400) THEN
		Curve_input:=TO_UINT(PWM_Y10_SET_Target1 - 400);
		IF(Curve_input>900) THEN
			Curve_input:=900;
		END_IF
		curve10(input:=REAL_TO_UINT(UINT_TO_REAL(Curve_input)*72.8),Zero:=FALSE,Full:=FALSE,
			   PAR_Progression:=Curve_Par,OutputEnable:=TRUE);
		PWM_Y10_SET:=PAR_Valve1_NegFull + REAL_TO_UINT(UINT_TO_REAL(curve10.Output)/72.8);
	ELSE
		PWM_Y10_SET:=0;
	END_IF
    //Y7 8 9 10范围限制
	IF(PWM_Y7_SET>1300)THEN
		PWM_Y7_SET :=1300;
	END_IF
	IF(PWM_Y8_SET>1300)THEN
		PWM_Y8_SET :=1300;
	END_IF
	IF(PWM_Y9_SET>1300)THEN
		PWM_Y9_SET :=1300;
	END_IF
	IF(PWM_Y10_SET>1300)THEN
		PWM_Y10_SET :=1300;
	END_IF
	
	IF(PWM_Y7_SET<=300)THEN
		PWM_Y7_SET :=0;
	END_IF
	IF(PWM_Y8_SET<=300)THEN
		PWM_Y8_SET :=0;
	END_IF
	IF(PWM_Y9_SET<=300)THEN
		PWM_Y9_SET :=0;
	END_IF
	IF(PWM_Y10_SET<=300)THEN
		PWM_Y10_SET :=0;
	END_IF
	
	
	DOH_Y56:=FALSE;
	PWM_Y33_SET_Target:=417;//110排量
	PWM_Y33_SET := PWM_Y33_SET_Target;
	//PWM_Y7_SET:=0;
	//PWM_Y9_SET:=0;
	//PWM_Y8_SET:=0;
	//PWM_Y10_SET:=0;
	PWM_Y1_SET:=0;//PWM_Y1_Target 直接给输出 去除中间变量
	PWM_Y2_SET:=0; //PWM_Y2_Target 

	PWM_Y39_SET_Target:=0;
	PWM_Y40_SET_Target:=0;
	RAMP19(
	IN:=WORD_TO_INT(PWM_Y39_SET_Target), 
	ASCEND:= R_RAMP_xiehe, 
	DESCEND:= F_RAMP_xiehe, 
	TIMEBASE:=TIMEBASE_xiehe , 
	RESET:=FALSE , 
	OUT=>(PWM_Y39_SET_Target1));
	IF(PWM_Y39_SET_Target1>=400) THEN
	Curve_input:=TO_UINT(PWM_Y39_SET_Target1 - 400);
	IF(Curve_input>900) THEN
		Curve_input:=900;
	END_IF
	curve19(input:=REAL_TO_UINT(UINT_TO_REAL(Curve_input)*72.8),Zero:=FALSE,Full:=FALSE,
		   PAR_Progression:=Curve_Par1,OutputEnable:=TRUE);
	PWM_Y39_SET:=PAR_Valve1_NegFull + REAL_TO_UINT(UINT_TO_REAL(curve19.Output)/72.8);
	ELSE
	PWM_Y39_SET:=0;
	END_IF


RAMP20(
	IN:=WORD_TO_INT(PWM_Y40_SET_Target), 
	ASCEND:= R_RAMP_xiehe, 
	DESCEND:= F_RAMP_xiehe, 
	TIMEBASE:=TIMEBASE_xiehe , 
	RESET:=FALSE , 
	OUT=>(PWM_Y40_SET_Target1));
IF(PWM_Y40_SET_Target1>=400) THEN
	Curve_input:=TO_UINT(PWM_Y40_SET_Target1 - 400);
	IF(Curve_input>900) THEN
		Curve_input:=900;
	END_IF
	curve20(input:=REAL_TO_UINT(UINT_TO_REAL(Curve_input)*72.8),Zero:=FALSE,Full:=FALSE,
		   PAR_Progression:=Curve_Par1,OutputEnable:=TRUE);
	PWM_Y40_SET:=PAR_Valve1_NegFull + REAL_TO_UINT(UINT_TO_REAL(curve20.Output)/72.8);
ELSE
	PWM_Y40_SET:=0;
END_IF
	
IF(PWM_Y39_SET>1300)THEN
	PWM_Y39_SET :=1300;
END_IF
IF(PWM_Y40_SET>1300)THEN
	PWM_Y40_SET :=1300;
END_IF

IF(PWM_Y39_SET<=300)THEN
	PWM_Y39_SET :=0;
END_IF
IF(PWM_Y40_SET<=300)THEN
	PWM_Y40_SET :=0;
END_IF

(*
	PWM_Y8_SET:=REAL_TO_UINT(INT_TO_REAL(PWM_JOYY_L_UP_1)/1000*(PAR_Valve1_PosFull-PAR_Valve1_NegFull)+PAR_Valve1_NegFull);
	PWM_Y10_SET:=REAL_TO_UINT(INT_TO_REAL(PWM_JOYY_L_UP_1)/1000*(PAR_Valve2_PosFull-PAR_Valve2_NegFull)+PAR_Valve2_NegFull);
	PWM_Y1_Target:=REAL_TO_UINT(INT_TO_REAL(PWM_JOYY_L_UP_1)/1000*(PAR_Y1_PosFull-PAR_Y1_NegFull)+PAR_Y1_NegFull);
	PWM_Y2_Target:=REAL_TO_UINT(INT_TO_REAL(PWM_JOYY_L_UP_1)/1000*(PAR_Y1_PosFull-PAR_Y2_NegFull)+PAR_Y2_NegFull);
*)
(*  //Y33输出处理
	IF PWM_Y33_SET>=PWM_Y33_SET_Target THEN
	PWM_Y33_SET := PWM_Y33_SET_Target;
	END_IF
		
	IF(PWM_Y33_SET<PWM_Y33_SET_Target) THEN
		PWM_Y33_SET:=REAL_TO_UINT(UINT_TO_REAL(PWM_Y33_SET)+JianGE6);
	END_IF
	
	IF DIL_SQ3 THEN
		PWM_Y33_SET:=0;
	END_IF
*)	
(*主泵功率控制*)

//区分发动机转速
MainPump_Pressure_Taget1450:=PAR_NegFull_x;
MainPump_Pressure_Taget1600:=PAR_PosFull_x;
MainPump_Pressure_Taget1750:=PAR_Zero_x;
IF EngineSpeedTarget<=1080 THEN SPEED_CASE:=1;
ELSIF EngineSpeedTarget>1080 AND EngineSpeedTarget<=1300 THEN SPEED_CASE:=2;
ELSIF EngineSpeedTarget>1300 AND EngineSpeedTarget<=1520 THEN SPEED_CASE:=3;
ELSIF EngineSpeedTarget>1520 AND EngineSpeedTarget<=1680 THEN SPEED_CASE:=4;
ELSIF EngineSpeedTarget>1680 AND EngineSpeedTarget<=1820 THEN SPEED_CASE:=5;
ELSIF EngineSpeedTarget>1820 THEN SPEED_CASE:=6;;END_IF
//不同转速下的发动机最大功率*)
CASE SPEED_CASE OF
1:  Enginer_Power:=135;
2:  Enginer_Power:=174;
3:  Enginer_Power:=200;
4:  Enginer_Power:=230;
5:  Enginer_Power:=250;
6:  Enginer_Power:=261;
END_CASE
//不同转速下的压力值
IF(CANO_Fubeng_Press>100)THEN
	CASE SPEED_CASE OF
	1:MainPump_Pressure_Taget:=MainPump_Pressure_Taget1000-HELIU_Press_Target1000;
	2:MainPump_Pressure_Taget:=MainPump_Pressure_Taget1200-HELIU_Press_Target1200;
	3:MainPump_Pressure_Taget:=MainPump_Pressure_Taget1450-HELIU_Press_Target1400;
	4:MainPump_Pressure_Taget:=MainPump_Pressure_Taget1600-HELIU_Press_Target1600;
	5:MainPump_Pressure_Taget:=MainPump_Pressure_Taget1750-HELIU_Press_Target1800;
	6:MainPump_Pressure_Taget:=MainPump_Pressure_Taget1900-HELIU_Press_Target1900;
	END_CASE
ELSE
	CASE SPEED_CASE OF
	1:MainPump_Pressure_Taget:=MainPump_Pressure_Taget1000;
	2:MainPump_Pressure_Taget:=MainPump_Pressure_Taget1200;
	3:MainPump_Pressure_Taget:=MainPump_Pressure_Taget1450;
	4:MainPump_Pressure_Taget:=MainPump_Pressure_Taget1600;
	5:MainPump_Pressure_Taget:=MainPump_Pressure_Taget1750;
	6:MainPump_Pressure_Taget:=MainPump_Pressure_Taget1900;
	END_CASE		
END_IF

IF( CANI_ECOSwitch) THEN
	CASE SPEED_CASE OF
	1:MainPump_Pressure_Taget:=MainPump_Pressure_Taget1000-ECO_Press_Target1000;
	2:MainPump_Pressure_Taget:=MainPump_Pressure_Taget1200-ECO_Press_Target1200;
	3:MainPump_Pressure_Taget:=MainPump_Pressure_Taget1450-ECO_Press_Target1400;
	4:MainPump_Pressure_Taget:=MainPump_Pressure_Taget1600-ECO_Press_Target1600;
	5:MainPump_Pressure_Taget:=MainPump_Pressure_Taget1750-ECO_Press_Target1800;
	6:MainPump_Pressure_Taget:=MainPump_Pressure_Taget1900-ECO_Press_Target1900;
	END_CASE
END_IF
MainPump_Pressure:=CANO_MainPUMP_Press1+CANO_MainPUMP_Press2;
//消除滤波
MainPump_Pressure_Subtract:= UINT_TO_INT(MainPump_Pressure-MainPump_Pressure_last1);


//大范围波动
IF MainPump_Pressure_Subtract>270 OR MainPump_Pressure_Subtract<-270 THEN
	Subtract:=TRUE;
ELSE
	Subtract:=FALSE;	
END_IF
	TIME_LvBo4(IN:=Subtract,PT:=T#10MS);
	
IF(TIME_LvBo4.Q)  AND (CANO_MainPUMP_Press1>210) THEN 
		MainPump_Pressure_ChangeBool1:=TRUE;
END_IF
	TIME_LvBo1(IN:=MainPump_Pressure_ChangeBool1,PT:=T#2S);
IF(TIME_LvBo1.Q) THEN
	MainPump_Pressure_ChangeBool1 :=FALSE;
END_IF

IF(MainPump_Pressure_ChangeBool1) AND (MainPump_Pressure>MainPump_Pressure_last1) THEN 
	MainPump_Pressure_last1:=MainPump_Pressure;
END_IF

//小范围波动
t_powertime:=TO_TIME(PAR_DeadBand_x);
IF (NOT MainPump_Pressure_ChangeBool1) THEN
	IF(MainPump_Pressure_Subtract>40 OR MainPump_Pressure_Subtract<-40)THEN 
		MainPump_Pressure_ChangeBool:=TRUE;
	ELSE
		MainPump_Pressure_ChangeBool:=FALSE;
	END_IF

	TIME_LvBo2(IN:=MainPump_Pressure_ChangeBool,PT:=t_powertime);
	IF(TIME_LvBo2.Q )THEN
		MainPump_Pressure_last1:=MainPump_Pressure;
	END_IF	
END_IF


IF PowerHead_move AND NOT(MainWinch_move) THEN
		JianGE2:=0.005;
ELSE
	IF(EngineSpeedTarget>1000 AND EngineSpeedTarget<1300)THEN
		JianGE2:=0.005;
	ELSE
		JianGE2:=0.005;
	END_IF
END_IF


IF MainPump_Pressure_last1>MainPump_Pressure_Taget THEN
	Pressure_Coe_Taget:=UINT_TO_REAL(MainPump_Pressure_Taget)/UINT_TO_REAL(MainPump_Pressure_last1);(*压力系数*)
ELSE
	Pressure_Coe_Taget:=1;
END_IF
Pressure_Coe := Pressure_Coe_Taget;


Pressure_Coe := 1;
IF MainPump_Pressure_last1>MainPump_Pressure_Taget  THEN
	IF(PWM_Y1_Target>=PAR_Y1_1_NegFull)THEN
		PWM_Y1_Target_OutPut:=REAL_TO_UINT(UINT_TO_REAL(PWM_Y1_Target-PAR_Y1_1_NegFull)*Pressure_Coe+PAR_Y1_1_NegFull);
	END_IF
	IF(PWM_Y2_Target>=PAR_Y1_1_NegFull)THEN
		PWM_Y2_Target_OutPut:=REAL_TO_UINT(UINT_TO_REAL(PWM_Y2_Target-PAR_Y1_1_NegFull)*Pressure_Coe+PAR_Y1_1_NegFull);
	END_IF
ELSE
	PWM_Y1_Target_OutPut:=PWM_Y1_Target;
	PWM_Y2_Target_OutPut:=PWM_Y2_Target;
END_IF

//PWM_Y1_Target_OutPut:=PWM_Y1_Target;
//PWM_Y2_Target_OutPut:=PWM_Y2_Target;
IF(EngineSpeedTarget>CANO_SPEED AND CANO_SPEED>400)THEN
	EngineSpeedSub:=EngineSpeedTarget - CANO_SPEED;
ELSE
	EngineSpeedSub:=0;
END_IF

IF(PWM_Y1_Target_OutPut<300)THEN PWM_Y1_Target_OutPut:=300;END_IF	
IF(PWM_Y2_Target_OutPut<300)THEN PWM_Y2_Target_OutPut:=300;END_IF

RAMP15_IN:=PWM_Y1_Target_OutPut;
RAMP16_IN:=PWM_Y2_Target_OutPut;
(*
IF MainWinch_move  OR  LeftMove_move OR RightMove_move THEN  
	TIMEBASE_pump:=T#1000MS;
	TIMEBASE_xiehe:=T#500MS;
ELSE
	TIMEBASE_pump:=T#400MS;
	TIMEBASE_xiehe:=T#200MS;
END_IF
t_PowerHead_move(IN:= MainWinch_move,PT:=T#2S);
IF t_PowerHead_move.Q THEN
	F_RAMP_pump:=x_t_PowerHead_move;
	R_RAMP_pump:=x2_t_PowerHead_move;
ELSE
	F_RAMP_pump:=1000;
	R_RAMP_pump:=300;
END_IF
*)
(*  12模式不需要斜坡
RAMP15(
	IN:=UINT_TO_INT(RAMP15_IN), 
	ASCEND:= 300, 
	DESCEND:= 300, 
	TIMEBASE:=T#1000MS , 
	RESET:=FALSE , 
	OUT=>(PWM_Y1_SET));
	
RAMP16(
	IN:=UINT_TO_INT(RAMP16_IN), 
	ASCEND:= 300, 
	DESCEND:= 300, 
	TIMEBASE:=T#1000MS , 
	RESET:=FALSE , 
	OUT=>(PWM_Y2_SET));

*)

	CASE SPEED_CASE OF
                1:F_RAMP_pump:=1500; R_RAMP_pump:=100;                  
                2: 		IF MainWinch_move AND (JiaYa_move OR CANO_JiayaPressure>80)  THEN    //3泵同时起压时，降低主泵的加载速度，避免掉速熄火
                                F_RAMP_pump:=1500; R_RAMP_pump:=100;
                        ELSE
                                F_RAMP_pump:=1500; R_RAMP_pump:=100;//从200降
                                IF  PWM_JOYY_L_UP>10 THEN
                                 F_RAMP_pump:=1500; R_RAMP_pump:=200;
                                END_IF
                        END_IF            
                3:
                        IF MainWinch_move AND (JiaYa_move OR CANO_JiayaPressure>80)  THEN    //3泵同时起压时，降低主泵的加载速度，避免掉速熄火
                                F_RAMP_pump:=1500; R_RAMP_pump:=150;
                        ELSE
                                F_RAMP_pump:=1500; R_RAMP_pump:=TO_INT(PAR_NegFull_y);
                                IF  PWM_JOYY_L_UP>10 THEN
                                 F_RAMP_pump:=1500; R_RAMP_pump:=300;
                                END_IF
                        END_IF                
                4:
                        IF MainWinch_move AND (JiaYa_move OR CANO_JiayaPressure>80)  THEN
                                F_RAMP_pump:=1500; R_RAMP_pump:=150;
                        ELSE
                                F_RAMP_pump:=1500; R_RAMP_pump:=TO_INT(PAR_PosFull_y);//从200降
                                IF  PWM_JOYY_L_UP>10 THEN
                                 F_RAMP_pump:=1500; R_RAMP_pump:=300;
                                END_IF
                        END_IF                                
                5:
                        IF MainWinch_move AND (JiaYa_move OR CANO_JiayaPressure>80)  THEN
                                F_RAMP_pump:=1500; R_RAMP_pump:=200;
                        ELSE
                                F_RAMP_pump:=1500; R_RAMP_pump:=TO_INT(PAR_Zero_y);
                                IF  PWM_JOYY_L_UP>10 THEN
                                 F_RAMP_pump:=1500; R_RAMP_pump:=300;
                                END_IF
                        END_IF                        
                6:		IF MainWinch_move AND (JiaYa_move OR CANO_JiayaPressure>80)  THEN
                                F_RAMP_pump:=1500; R_RAMP_pump:=200;
                        ELSE
                                F_RAMP_pump:=1500; R_RAMP_pump:=200;
                                IF  PWM_JOYY_L_UP>10 THEN
                                 F_RAMP_pump:=1500; R_RAMP_pump:=300;
                                END_IF
                        END_IF	
	END_CASE
(******斜坡增步长300 斜坡降步长300->400*****)	
RAMP15(
	IN:=UINT_TO_INT(RAMP15_IN), 
	ASCEND:= R_RAMP_pump, 
	DESCEND:= 1500, 
	TIMEBASE:=T#1000MS , 
	RESET:=FALSE , 
	OUT=>(PWM_Y1_SET));
(******减斜坡300->400*****)	
RAMP16(
	IN:=UINT_TO_INT(RAMP16_IN), 
	ASCEND:= R_RAMP_pump, 
	DESCEND:= 1500, 
	TIMEBASE:=T#1000MS , 
	RESET:=FALSE , 
	OUT=>(PWM_Y2_SET));

IF (NOT Rotation_move) AND (NOT MainWinch_move) AND (NOT PowerHead_move)
		AND (NOT JiaYa_move) AND (NOT ViceWinch_move)
		AND (NOT LeftMove_move) AND (NOT RightMove_move)  THEN
	PWM_Y1_Target:=0;
	PWM_Y2_Target:=0;
END_IF

IF PWM_Y1_SET<TO_INT(PAR_Y1_1_NegFull )THEN
	PWM_Y1_SET:=TO_INT(PAR_Y1_1_NegFull);
END_IF

IF PWM_Y2_SET<TO_INT(PAR_Y1_1_NegFull )THEN
	PWM_Y2_SET:=TO_INT(PAR_Y1_1_NegFull);
END_IF

IF(PWM_Y1_SET>1000) THEN
	PWM_Y1_SET := 300;
END_IF

IF(PWM_Y2_SET>1000) THEN
	PWM_Y2_SET := 300;
END_IF

END_PROGRAM

// StandardPLC/Application/SaveEngine/SaveEngineMode_9
PROGRAM SaveEngineMode_9
VAR
DI_PWM_JOYX_L: BOOL;
	DI_PWM_JOYY_L: BOOL;
	DI_PWM_JOYX_R: BOOL;
	DI_PWM_JOYY_R: BOOL;
	DI_PWM_JOY_Jiao_R: BOOL;
	DI_PWM_JOY_Jiao_L: BOOL;
	Rotation_move: BOOL;
	MainWinch_move:BOOL;
	PowerHead_move:BOOL;
	JiaYa_move: BOOL;
	LvZhang_move: BOOL;
	BianFu_move:BOOL;
	ViceWinch_move: BOOL;
	LeftMove_move:BOOL;
	RightMove_move:BOOL;
	SPEED_CASE:USINT;
	Enginer_Power:UINT;
	
	PWM_Y1_Target: UINT;	
	PWM_Y2_Target: UINT;	
	
	PWM_Y1_Target_MAX: UINT;
	PWM_Y2_Target_MAX: UINT;
	Hydraulic_Power2:UINT;
	Hydraulic_Power1:UINT;
	Hydraulic_Power:UINT;
	Enginer_Rat: UINT;
	MainPump_Pressure_Taget:UINT;
	Coe_valve: REAL;	
	MainPump_Pressure: UINT;
	Pressure_Coe: REAL;
	PWM_Y1_Target_1: UINT;
	Single_move:BOOL;
	PWM_Y1_Target_OutPut: UINT;
	PWM_Y2_Target_OutPut: UINT;
	PWM_Y34_SET_Target: UINT:=0;
	PWM_Y33_SET_Target: UINT:=1100;
	

	DonglitouBlink:BLINK;
	DonglitouBlink_biaozhi:BOOL;
	DOH_Y50_1: BOOL;
	Rotation_late:TOF;
	MainPump_Pressure_Taget1000:UINT:=220;
	MainPump_Pressure_Taget1200:UINT:=360;
	MainPump_Pressure_Taget1450:UINT:=420;
	MainPump_Pressure_Taget1600:UINT:=420;
	MainPump_Pressure_Taget1750:UINT:=400;
	MainPump_Pressure_Taget1900:UINT:=360;
	Pressure_Coe_Taget: REAL;
	JianGE1: REAL:=1;
	JianGE2: REAL:=0.005;
	JianGE3: REAL:=3;
	TIME_100ms:TON;
	MainPump_Pressure_last: UINT;
	MainPump_Pressure_last1: UINT;
	TIME_LvBo1:TON;
	TIME_LvBo2:TON;
	TIME_LvBo3:TON;
	MainPump_Pressure_Subtract: INT;
	MainPump_Pressure_ChangeBool: BOOL;
	MainPump_Pressure_ChangeBool1:BOOL;
	PWM_Y2_Target_fuhe: UINT;
	PWM_Y1_Target_fuhe: UINT;
	EngineSpeedSub: UINT;
	PWM_Y23_SET_Taget: UINT;
	PWM_Y24_SET_Taget: UINT;
	CANO_DonglitouPressure_last: UINT;
	DonglitouPressureSub:INT;
	DonglitouPressure_ChangeBool: BOOL;
	JieSuoBool: BOOL;
	ECO_Press_Target1000: UINT:=50;
	ECO_Press_Target1200: UINT:=50;
	ECO_Press_Target1400: UINT:=50;
	ECO_Press_Target1600: UINT:=50;
	ECO_Press_Target1800: UINT:=50;
	ECO_Press_Target1900: UINT:=50;
	
	HELIU_Press_Target1000: UINT:=80;
	HELIU_Press_Target1200: UINT:=80;
	HELIU_Press_Target1400: UINT:=80;
	HELIU_Press_Target1600: UINT:=80;
	HELIU_Press_Target1800: UINT:=80;
	HELIU_Press_Target1900: UINT:=80;
	PWM_Y2_Target_P: UINT;
	PWM_JOY_P_W: UINT;
	XISHU1: REAL:=0.6;
	BiaoZHI_MainWinchUp: BOOL;
	JianGE6:REAL:=2;
	PWM_Y5_SET_Target: UINT;
	PWM_Y6_SET_Target: UINT;
	PWM_Y15_SET_Target: UINT;
	PWM_Y16_SET_Target: UINT;
	PWM_Y5_SET_Target1: INT;
	PWM_Y6_SET_Target1: INT;
	PWM_Y15_SET_Target1: INT;
	PWM_Y16_SET_Target1: INT;
	PWM_Y8_SET_Target: UINT;
	PWM_Y10_SET_Target: UINT;
	PWM_Y7_SET_Target: UINT;
	PWM_Y9_SET_Target: UINT;
	PWM_Y8_SET_Target1: INT;
	PWM_Y10_SET_Target1: INT;
	PWM_Y7_SET_Target1: INT;
	PWM_Y9_SET_Target1: INT;
	JianGE7: UINT:=20;
	JianGE8: UINT:=3;
	PWM_Y39_SET_Target: UINT;
	PWM_Y40_SET_Target: UINT;
	ABS_JOY_1: INT;
	PWM_Y61_SET_Tatget: UINT;
	PWM_Y12_SET_Tatget: UINT;
	PWM_Y14_SET_Tatget: UINT;
	PWM_Y60_SET_Tatget: UINT;
	PWM_Y11_SET_Tatget: UINT;
	PWM_Y13_SET_Tatget: UINT;
	PWM_Y61_SET_Tatget1: INT;
	PWM_Y12_SET_Tatget1: INT;
	PWM_Y14_SET_Tatget1: INT;
	PWM_Y60_SET_Tatget1: INT;
	PWM_Y11_SET_Tatget1: INT;
	PWM_Y13_SET_Tatget1: INT;
	JianGE10: UINT:=25;
	yyyy: UINT;
	TIME_200ms:TON;
	TIME_400ms:TON;
	CANI_JOYX_R_last:UINT;
	Sub_Joyx_r: INT;
	Joyx_change_bool: BOOL;
	JianGE12: UINT:=30;
	Sub_Joyx_r_1: INT;
	BIAOzhi1: BOOL;
	R_TRIG_1:R_TRIG;
	R_TRIG_BOOL: BOOL;
	JianGE22: REAL;
	
	
	curve:curve_quxian;
	curve1:curve_quxian;
	curve2:curve_quxian;
	curve3:curve_quxian;
	curve4:curve_quxian;
	curve5:curve_quxian;
	curve6:curve_quxian;
	curve7:curve_quxian;
	curve8:curve_quxian;
	curve9:curve_quxian;
	curve10:curve_quxian;
	curve11:curve_quxian;
	curve12:curve_quxian;
	curve13:curve_quxian;
	curve14:curve_quxian;
	curve19:curve_quxian;
	curve20:curve_quxian;
	COUNTER : INT;
	JianGE13: UINT:=40;
	JianGE14: UINT:=40;
	RAMP:RAMP_INT;
	RAMP1:RAMP_INT;
	RAMP2:RAMP_INT;
	RAMP3:RAMP_INT;
	R_RAMP:INT:=400;
	F_RAMP:INT:=250;
	TIMEBASE:TIME:=T#200MS;
	PWM_Y7_SET_Target111: INT;
	YYYYYYY:BOOL;
	JIANGE1111: INT:=20;
	
	RAMP4:RAMP_INT;
	RAMP5:RAMP_INT;
	RAMP6:RAMP_INT;
	RAMP7:RAMP_INT;
	RAMP8:RAMP_INT;
	RAMP9:RAMP_INT;
	RAMP10:RAMP_INT;
	RAMP11:RAMP_INT;
	RAMP12:RAMP_INT;
	RAMP13:RAMP_INT;
	RAMP14:RAMP_INT;
	RAMP15:RAMP_INT;
	RAMP16:RAMP_INT;
	RAMP17:RAMP_INT;
	RAMP18:RAMP_INT;
	RAMP19:RAMP_INT;
	RAMP20:RAMP_INT;
	RAMP21:RAMP_INT;
	RAMP22:RAMP_INT;
	RAMP23:RAMP_INT;
	RAMP24:RAMP_INT;
	PWM_Y23_SET_Taget1:INT;
	PWM_Y24_SET_Taget1:INT;
	PWM_Y18_SET_Taget1:INT;
	PWM_Y18_SET_Taget:UINT;
	ASCEND_value2:INT;
	//2023 01 13 增加
	//行走动作斜坡值
	R_RAMP_traval:INT:=800;
	F_RAMP_traval:INT:=400;
	TIMEBASE_traval:TIME:=T#200MS;
	//动力头动作斜坡值
	R_RAMP_ratate:INT:=800;
	F_RAMP_ratate:INT:=800;
	TIMEBASE_ratate:TIME:=T#100MS;
	//主卷扬动作斜坡值
	R_RAMP_mainwinch:INT:=800;
	F_RAMP_mainwinch_up:INT:=400;
	F_RAMP_mainwinch_down:INT:=400;
	TIMEBASE_mainwinch:TIME:=T#200MS;
	//主泵排量斜坡值
	R_RAMP_pump:INT:=300;
	F_RAMP_pump:INT:=1000;
	TIMEBASE_pump:TIME:=T#1000MS;
	//卸荷阀斜坡值
	R_RAMP_xiehe:INT:=500;
	F_RAMP_xiehe:INT:=400;
	TIMEBASE_xiehe:TIME:=T#500MS;
	
	//直线阀斜坡值
	R_RAMP_zhixian:INT:=800;
	F_RAMP_zhixian:INT:=800;
	TIMEBASE_zhixian:TIME:=T#300MS;
		
	Subtract: BOOL;
	TIME_LvBo4:TON;
	Curve_input:UINT;
	Curve_Par: SINT:=0;
	Curve_Par1: SINT:=0;
	Move_JOY_FUHE: UINT;
	PWM_JOY_Jiao_L_UP1:UINT;
	PWM_JOY_Jiao_L_DOWN1:UINT;
	PWM_JOY_Jiao_R_UP1:UINT;
	PWM_JOY_Jiao_R_DOWN1:UINT;
	
	PWM_JOYX_R_UP_a:UINT;
	PWM_JOYX_R_UP_b:UINT;
	
	PWM_JOYX_R_DOWN_a:UINT;
	PWM_JOYX_R_DOWN_b:UINT;
	
	PWM_JOYY_L_DOWN_a:UINT;
	PWM_JOYY_L_DOWN_b:UINT;
	
	PWM_JOYY_L_UP_a:UINT;
	PWM_JOYY_L_UP_b:UINT;
	aaaa:UINT:=500;
	
	JOY_PAOTU:BOOL;
	
	JOY_PAOTU_tiaojian:BOOL;
	TIME_1000_1ms:ton;
	tempbool:BOOL;
	CANI_JOYX_R_last2:UINT;
	Sub_Joyx_r2:INT;
	JianGE11:REAL:=2;
	JianGE21:uint:=10;
	END_IFc: INT;
	x1:UINT:=8;
	x2:UINT:=8;
	PWM_JOY_JIAO:UINT;
	PWM_Y39_SET1:UINT;
	PWM_Y40_SET1:UINT;
	aaa: INT;
	TIME_50ms:TON;
	TIME_55ms:TOF;
	TIME_2000ms:TOF;
	start_move: BOOL;
	T1:TIME;
	TEMP1:UINT;
	X3: INT;
	X4: INT;
	liandong:BOOL;
	PWM_Y9_SET1:INT;
	PWM_Y10_SET1:INT;
	PWM_Y13_SET1:INT;
	PWM_Y14_SET1:INT;
	yanchi1:BOOL;
	yanchi_ton1:ton;
	RAMP15_IN:UINT;
	RAMP16_IN:UINT;
	Rtrig_d1:R_TRIG;
	Rtrig_d2:R_TRIG;
	
	Rtrig_DongLiTou1:R_TRIG;
	Rtrig_DongLiTou2:R_TRIG;
	Count_TIMES_Fanzhuan: UINT;
	Count_TIMES_Zhengzhuan: UINT;
	TIME_1000ms:TON;
	TIME_1000ms_TP:TON;
	Count_TIMES_Fanzhuan_LAST: UINT;
	Count_TIMES_Zhengzhuan_LAST: UINT;
	Paotu_Modle: BOOL;
	PaoTU_biaozhi: BOOL;
	TIMEBASE_D: TIME;
	PWM_Y39_SET_Target1:INT;
	PWM_Y40_SET_Target1:INT;
	PWM_Y37_SET_Target:UINT;
	PWM_Y17_SET2:UINT;
	t_PowerHead_move:TON;
	x_t_PowerHead_move:INT:=10;//100-10
	x2_t_PowerHead_move:INT:=10;//100-10
	P_value:REAL;//动力头反转+主卷上提时的分流系数
	PWM_JOY_P:UINT;
	PWM_JOY_P1:UINT;
	PWM_JOY_P2:UINT;
	PWM_JOY_P3:UINT;
	PWM_JOY_P4:UINT;
	ASCEND_value:INT;
	ftp1:INT:=500;
	ftp2:INT:=100;
	t_powertime:TIME;
	
	P25_Flag:BOOL;
	P27_Flag:BOOL;
	P29_Flag:BOOL;
	P31_Flag:BOOL;
	PressLvBo_TON:TON;
	PressLvBo_TON1: TON;
	PressLvBo_TON2: TON;
	PressLvBo_TON3: TON;
	test: BYTE;
	testpaotu: UINT := 450;
END_VAR

//动力头反转与主卷上提时的分流系数值
(*IF CANO_ZhuJuanPressure<=100 THEN
	P_value:=TO_REAL(PAR_KI+40)/100.0;
ELSIF CANO_ZhuJuanPressure>100 AND  CANO_ZhuJuanPressure<=200 THEN
	P_value:=TO_REAL(PAR_KI+20)/100.0;
ELSE
	P_value:=TO_REAL(PAR_KI)/100;
END_IF*)
GVL_SaveEngine.Y72OutPutState:=0;
GVL_SaveEngine.Y71OutPutState:=0;
GVL_SaveEngine.Y73:=0;
P_value:=TO_REAL(PAR_KI)/100;  //出厂值设定为35
//喇叭
IF DI_LHandle_SB5 THEN
	DOH_Y59:=TRUE;
ELSE
	DOH_Y59:=FALSE;
END_IF
//延时断电
TIME_2000ms(IN:=DIH_power3,PT:=T#2S);
IF(TIME_2000ms.Q)THEN
	DOH_YS3:=TRUE;
ELSE
	DOH_YS3:=FALSE;
END_IF

//主卷上限位及解锁
IF(DI_LHandle_SB1 AND (NOT CANI_WorkModeSwitch))THEN
	JieSuoBool:=TRUE;
ELSE
	JieSuoBool:=FALSE;	
END_IF

IF DIL_SQ4 THEN
	IF(NOT JieSuoBool) THEN
		PWM_JOYY_L_DOWN:=0;
	END_IF
END_IF

//主卷下限位及解锁
//主卷下放限制
IF( CANO_MainWinchTension*100<PAR_MainWinchLaLi_Low) AND (NOT DI_LHandle_SB1) AND (CANI_WorkModeSwitch)THEN
	PWM_JOYY_L_UP:=0;
END_IF

TIME_50ms(in:=start_move,pt:=T1);
TIME_55ms(in:=start_move,pt:=T#500MS);
IF( LeftMove_move OR  RightMove_move  OR   MainWinch_move OR PowerHead_move OR ViceWinch_move )THEN
	start_move:=TRUE;
ELSE
	start_move:=FALSE;
END_IF
	 


IF NOT DIL_SQ3 THEN(*先导控制输入*)
	IF PWM_JOYX_L_UP>10 OR PWM_JOYX_L_DOWN>10 THEN  DI_PWM_JOYX_L := TRUE;ELSE DI_PWM_JOYX_L:=FALSE;END_IF(*左手柄左右动作*)
	IF PWM_JOYY_L_UP>10 OR PWM_JOYY_L_DOWN>10 THEN  DI_PWM_JOYY_L := TRUE;ELSE DI_PWM_JOYY_L:=FALSE;END_IF(*左手柄前后动作*)
	IF PWM_JOYX_R_UP>10 OR PWM_JOYX_R_DOWN>10 THEN  DI_PWM_JOYX_R := TRUE;ELSE DI_PWM_JOYX_R:=FALSE;END_IF(*右手柄左右动作*)
	IF PWM_JOYY_R_UP>10 OR PWM_JOYY_R_DOWN>10 THEN  DI_PWM_JOYY_R := TRUE;ELSE DI_PWM_JOYY_R:=FALSE;END_IF(*右手柄前后动作*)
	IF PWM_JOY_Jiao_L_UP>10 OR PWM_JOY_Jiao_L_DOWN>10 THEN  DI_PWM_JOY_Jiao_L:= TRUE;ELSE DI_PWM_JOY_Jiao_L:=FALSE;END_IF(*左脚踏前后动作*)
	IF PWM_JOY_Jiao_R_UP>10 OR PWM_JOY_Jiao_R_DOWN>10 THEN  DI_PWM_JOY_Jiao_R := TRUE;ELSE DI_PWM_JOY_Jiao_R:=FALSE;END_IF(*左脚踏左右动作*)
ELSE
	DI_PWM_JOYX_L:=FALSE;
	DI_PWM_JOYY_L:=FALSE;
	DI_PWM_JOYX_R:=FALSE;
	DI_PWM_JOYY_R:=FALSE;
	DI_PWM_JOY_Jiao_L:=FALSE;
	DI_PWM_JOY_Jiao_R:=FALSE;
END_IF

(*动作标志*)
IF DI_PWM_JOYY_L THEN MainWinch_move:=TRUE; ELSE MainWinch_move:=FALSE;END_IF(*主卷扬动作*)
IF DI_PWM_JOYX_L THEN Rotation_move:=TRUE; ELSE Rotation_move:=FALSE;END_IF(*回转动作*)
IF CANI_WorkModeSwitch THEN   (*作业挡情况下*)
	IF DI_PWM_JOYX_R THEN PowerHead_move:=TRUE;ELSE PowerHead_move:=FALSE;END_IF(*动力头回转动作*)
	IF DI_PWM_JOYY_R THEN JiaYa_move:=TRUE;ELSE JiaYa_move:=FALSE;END_IF(*动力头加压动作*)
	LvZhang_move:=FALSE;
	BianFu_move:=FALSE;
	ViceWinch_move:=FALSE;
	LeftMove_move:=FALSE;
	RightMove_move:=FALSE;
ELSE   (*调整档状态*)
	IF DI_PWM_JOYX_R THEN  LvZhang_move:=TRUE;ELSE LvZhang_move:=FALSE;END_IF(*L履带、张紧、支腿动作,M4阀*)
	(*LeftMove_move:=DI_PWM_JOY_Jiao_L;(*左行走动作*)
	RightMove_move:=DI_PWM_JOY_Jiao_R;*)(*右行走动作*)
	IF( PWM_JOY_Jiao_L_UP1>10 OR PWM_JOY_Jiao_L_DOWN1>10)  AND  DI_PWM_JOY_Jiao_L THEN
		LeftMove_move:=TRUE;
	ELSE
		LeftMove_move:=FALSE;
	END_IF
	IF( PWM_JOY_Jiao_R_UP1>10 OR PWM_JOY_Jiao_R_DOWN1>10)  AND  DI_PWM_JOY_Jiao_R THEN
		RightMove_move:=TRUE;
	ELSE
		RightMove_move:=FALSE;
	END_IF

	IF  DI_RHandle_SB5 THEN
		ViceWinch_move:=FALSE;
		IF  DI_PWM_JOYY_R  THEN BianFu_move:=TRUE;ELSE BianFu_move:=FALSE;END_IF(*变幅动作M4阀*)
	ELSE
		BianFu_move:=FALSE;
		IF DI_PWM_JOYY_R  THEN ViceWinch_move:=TRUE;ELSE ViceWinch_move:=FALSE;END_IF(*副卷扬动作M4阀*)
	END_IF
	PowerHead_move:=FALSE;
	JiaYa_move:=FALSE;
END_IF


(****主阀单动作标志****)
	IF (NOT MainWinch_move) AND (NOT PowerHead_move) AND (ViceWinch_move) THEN
		Single_move:=TRUE;
	ELSE
		Single_move:=FALSE;
	END_IF
	
//先导控制
IF(NOT DIL_SQ3) AND NOT VarGpsSystemLockedState THEN
	DOH_Y51:=TRUE;
ELSE
	DOH_Y51:=FALSE;
END_IF

//行走动作
(*脚踏阀偏差*)
IF   ((PWM_JOY_Jiao_L_UP-PWM_JOY_Jiao_R_UP)<200 OR(PWM_JOY_Jiao_R_UP-PWM_JOY_Jiao_L_UP)<200) THEN
	PWM_JOY_Jiao_L_UP1:=MAX(PWM_JOY_Jiao_L_UP,PWM_JOY_Jiao_R_UP);
	PWM_JOY_Jiao_R_UP1:=MAX(PWM_JOY_Jiao_L_UP,PWM_JOY_Jiao_R_UP);
ELSE
	PWM_JOY_Jiao_L_UP1:=PWM_JOY_Jiao_L_UP;
	PWM_JOY_Jiao_R_UP1:=PWM_JOY_Jiao_R_UP;
END_IF
IF   ((PWM_JOY_Jiao_L_DOWN-PWM_JOY_Jiao_R_DOWN)<200  OR  (PWM_JOY_Jiao_R_DOWN-PWM_JOY_Jiao_L_DOWN)<200 ) THEN
	PWM_JOY_Jiao_L_DOWN1:=MAX(PWM_JOY_Jiao_L_DOWN,PWM_JOY_Jiao_R_DOWN);
	PWM_JOY_Jiao_R_DOWN1:=MAX(PWM_JOY_Jiao_L_DOWN,PWM_JOY_Jiao_R_DOWN);
ELSE
	PWM_JOY_Jiao_L_DOWN1:=PWM_JOY_Jiao_L_DOWN;
	PWM_JOY_Jiao_R_DOWN1:=PWM_JOY_Jiao_R_DOWN;
END_IF

PWM_JOY_JIAO:=MAX(PWM_JOY_Jiao_L_UP1,PWM_JOY_Jiao_R_UP1,PWM_JOY_Jiao_L_DOWN1,PWM_JOY_Jiao_R_DOWN1);
liandong:=FALSE;
(*左行走*)
(*泵1   Y1   Y39控制右行走   Y15  16 *)
(*泵2   Y2 Y40 控制左行走    Y5  Y6*)
IF LeftMove_move THEN
	IF PWM_JOY_Jiao_L_UP1>10 THEN
		PWM_Y2_Target:=REAL_TO_UINT(UINT_TO_REAL(PWM_JOY_Jiao_L_UP1)/1000*(PAR_Y1_1_PosFull-PAR_Y1_1_NegFull)+PAR_Y1_1_NegFull);
		PWM_Y5_SET_Target:=REAL_TO_UINT(UINT_TO_REAL(PWM_JOY_Jiao_L_UP1)/1000*(PAR_Valve2_PosFull-PAR_Valve2_NegFull)+PAR_Valve2_NegFull);
		PWM_Y6_SET_Target:=0;	
	ELSIF PWM_JOY_Jiao_L_DOWN1>10 THEN
		PWM_Y2_Target:=REAL_TO_UINT(UINT_TO_REAL(PWM_JOY_Jiao_L_DOWN1)/1000*(PAR_Y1_1_PosFull-PAR_Y1_1_NegFull)+PAR_Y1_1_NegFull);
		PWM_Y6_SET_Target:=REAL_TO_UINT(UINT_TO_REAL(PWM_JOY_Jiao_L_DOWN1)/1000*(PAR_Valve2_PosFull-PAR_Valve2_NegFull)+PAR_Valve2_NegFull);
		PWM_Y5_SET_Target:=0;		
	END_IF
ELSE
	PWM_Y5_SET_Target:=0;
	PWM_Y6_SET_Target:=0;
END_IF
(*右行走*)
IF RightMove_move  THEN
	IF PWM_JOY_Jiao_R_UP1>10 THEN
		PWM_Y1_Target:=REAL_TO_UINT(UINT_TO_REAL(PWM_JOY_Jiao_R_UP1)/1000*(PAR_Y1_1_PosFull-PAR_Y1_1_NegFull)+PAR_Y1_1_NegFull);
		PWM_Y15_SET_Target:=REAL_TO_UINT(UINT_TO_REAL(PWM_JOY_Jiao_R_UP1)/1000*(PAR_Valve1_PosFull-PAR_Valve1_NegFull)+PAR_Valve1_NegFull);
		PWM_Y16_SET_Target:=0;
	
	ELSIF PWM_JOY_Jiao_R_DOWN1>10 THEN
		PWM_Y1_Target:=REAL_TO_UINT(UINT_TO_REAL(PWM_JOY_Jiao_R_DOWN1)/1000*(PAR_Y1_1_PosFull-PAR_Y1_1_NegFull)+PAR_Y1_1_NegFull);
		PWM_Y16_SET_Target:=REAL_TO_UINT(UINT_TO_REAL(PWM_JOY_Jiao_R_DOWN1)/1000*(PAR_Valve1_PosFull-PAR_Valve1_NegFull)+PAR_Valve1_NegFull);
		PWM_Y15_SET_Target:=0;
		
	END_IF
ELSE
	PWM_Y15_SET_Target:=0;
	PWM_Y16_SET_Target:=0;
END_IF

	//如有必要，可根据行走阀开关大小调整斜坡值
(*	IF(PWM_Y5_SET<1000  AND  PWM_Y5_SET>=900)THEN
			R_RAMP_traval:=100;
	ELSIF(PWM_Y5_SET<900 AND PWM_Y5_SET>=780)THEN
			R_RAMP_traval:=10;
	ELSE
			R_RAMP_traval:=250;
	END_IF
		
	IF(PWM_Y6_SET<1000  AND  PWM_Y6_SET>=900)THEN
			F_RAMP_traval:=100;		
	ELSIF(PWM_Y6_SET<900 AND PWM_Y6_SET>750 )THEN
			F_RAMP_traval:=15;
	ELSE
			F_RAMP_traval:=250;
	END_IF*)
	
(*行走动作缓冲*)
RAMP11(
	IN:=WORD_TO_INT(PWM_Y5_SET_Target), 
	ASCEND:= R_RAMP_traval, 
	DESCEND:= F_RAMP_traval, 
	TIMEBASE:=TIMEBASE_traval , 
	RESET:=FALSE , 
	OUT=>(PWM_Y5_SET_Target1));
IF(PWM_Y5_SET_Target1>=400) THEN
	Curve_input:=TO_UINT(PWM_Y5_SET_Target1 - 400);
	IF(Curve_input>900) THEN
		Curve_input:=900;
	END_IF
	curve11(input:=REAL_TO_UINT(UINT_TO_REAL(Curve_input)*72.8),Zero:=FALSE,Full:=FALSE,
		   PAR_Progression:=Curve_Par1,OutputEnable:=TRUE);
	PWM_Y5_SET:=PAR_Valve1_NegFull + REAL_TO_UINT(UINT_TO_REAL(curve11.Output)/72.8);
ELSE
	PWM_Y5_SET:=0;
END_IF

RAMP12(
	IN:=WORD_TO_INT(PWM_Y6_SET_Target), 
	ASCEND:= R_RAMP_traval, 
	DESCEND:= F_RAMP_traval, 
	TIMEBASE:=TIMEBASE_traval , 
	RESET:=FALSE , 
	OUT=>(PWM_Y6_SET_Target1));
IF(PWM_Y6_SET_Target1>=400) THEN
	Curve_input:=TO_UINT(PWM_Y6_SET_Target1 - 400);
	IF(Curve_input>900) THEN
		Curve_input:=900;
	END_IF
	curve12(input:=REAL_TO_UINT(UINT_TO_REAL(Curve_input)*72.8),Zero:=FALSE,Full:=FALSE,
		   PAR_Progression:=Curve_Par1,OutputEnable:=TRUE);
	PWM_Y6_SET:=PAR_Valve1_NegFull + REAL_TO_UINT(UINT_TO_REAL(curve12.Output)/72.8);
ELSE
	PWM_Y6_SET:=0;
END_IF

RAMP13(
	IN:=WORD_TO_INT(PWM_Y15_SET_Target), 
	ASCEND:= R_RAMP_traval, 
	DESCEND:= F_RAMP_traval, 
	TIMEBASE:=TIMEBASE_traval , 
	RESET:=FALSE , 
	OUT=>(PWM_Y15_SET_Target1));
IF(PWM_Y15_SET_Target1>=400) THEN
	Curve_input:=TO_UINT(PWM_Y15_SET_Target1 - 400);
	IF(Curve_input>900) THEN
		Curve_input:=900;
	END_IF
	curve13(input:=REAL_TO_UINT(UINT_TO_REAL(Curve_input)*72.8),Zero:=FALSE,Full:=FALSE,
		   PAR_Progression:=Curve_Par1,OutputEnable:=TRUE);
	PWM_Y15_SET:=PAR_Valve1_NegFull + REAL_TO_UINT(UINT_TO_REAL(curve13.Output)/72.8);
ELSE
	PWM_Y15_SET:=0;
END_IF

RAMP14(
	IN:=WORD_TO_INT(PWM_Y16_SET_Target), 
	ASCEND:= R_RAMP_traval, 
	DESCEND:= F_RAMP_traval, 
	TIMEBASE:=TIMEBASE_traval , 
	RESET:=FALSE , 
	OUT=>(PWM_Y16_SET_Target1));
IF(PWM_Y16_SET_Target1>=400) THEN
	Curve_input:=TO_UINT(PWM_Y16_SET_Target1 - 400);
	IF(Curve_input>900) THEN
		Curve_input:=900;
	END_IF
	curve14(input:=REAL_TO_UINT(UINT_TO_REAL(Curve_input)*72.8),Zero:=FALSE,Full:=FALSE,
		   PAR_Progression:=Curve_Par1,OutputEnable:=TRUE);
	PWM_Y16_SET:=PAR_Valve1_NegFull + REAL_TO_UINT(UINT_TO_REAL(curve14.Output)/72.8);
ELSE
	PWM_Y16_SET:=0;
END_IF


(*直线行走*)
(*IF(  DIH_SA19)THEN
	IF (PWM_JOY_Jiao_L_UP1>10  AND PWM_JOY_Jiao_R_UP1>10) OR ( PWM_JOY_Jiao_L_DOWN1>10 AND PWM_JOY_Jiao_R_DOWN1>10)THEN
		PWM_Y37_SET_Target:=800;  //开环  占控比   0-1000
	ELSE
		PWM_Y37_SET_Target:=0;
	END_IF
ELSE
	PWM_Y37_SET_Target:=0;
END_IF

IF((LeftMove_move OR RightMove_move)AND MainWinch_move)THEN
	PWM_Y1_Target:=REAL_TO_UINT(UINT_TO_REAL(PWM_JOY_JIAO)/1000*(PAR_Y2_PosFull-PAR_Y2_NegFull)+PAR_Y2_NegFull);
	PWM_Y2_Target:=0;
	PWM_Y37_SET_Target:=800;
END_IF*)
(*直线行走*)//Y2  Y40   行走阀
IF DIH_SA19 THEN
	PWM_Y37_SET_Target:=800;
	PWM_Y1_Target:=0;
ELSE
	PWM_Y37_SET_Target:=0;
END_IF

IF((LeftMove_move OR RightMove_move)AND MainWinch_move)THEN
	PWM_Y2_Target:=REAL_TO_UINT(UINT_TO_REAL(PWM_JOY_JIAO)/1000*(PAR_Y2_PosFull-PAR_Y2_NegFull)+PAR_Y2_NegFull);
	PWM_Y1_Target:=0;
	PWM_Y37_SET_Target:=800;
END_IF


RAMP21(
	IN:=UINT_TO_INT(PWM_Y37_SET_Target), 
	ASCEND:= R_RAMP_zhixian, 
	DESCEND:= F_RAMP_zhixian, 
	TIMEBASE:=TIMEBASE_zhixian , 
	RESET:=FALSE , 
	OUT=>(PWM_Y37_SET));


IF(PWM_JOYX_R_UP<=500)THEN
	PWM_JOYX_R_UP_a:=PWM_JOYX_R_UP;
	PWM_JOYX_R_UP_b:=0;
ELSE
	PWM_JOYX_R_UP_a:=500;
	PWM_JOYX_R_UP_b:=PWM_JOYX_R_UP-500;
END_IF

IF(PWM_JOYX_R_DOWN<=500)THEN
	PWM_JOYX_R_DOWN_a:=PWM_JOYX_R_DOWN;
	PWM_JOYX_R_DOWN_b:=0;
ELSE
	PWM_JOYX_R_DOWN_a:=500;
	PWM_JOYX_R_DOWN_b:=PWM_JOYX_R_DOWN-500;
END_IF

	
(*单动力头动作*)
IF (NOT MainWinch_move) AND(PowerHead_move) AND(NOT DI_RHandle_SB6) THEN
	IF PWM_JOYX_R_UP>10 THEN//动力头反转
			PWM_Y1_Target:=REAL_TO_UINT(UINT_TO_REAL(PWM_JOYX_R_UP)/1000*(PAR_Y1_PosFull-PAR_Y1_NegFull)+PAR_Y1_NegFull);			
			PWM_Y2_Target:=REAL_TO_UINT(UINT_TO_REAL(PWM_JOYX_R_UP_b)/500*(PAR_Y2_PosFull-PAR_Y2_NegFull)+PAR_Y2_NegFull);
		IF(DIH_SA18)THEN
			PWM_Y1_Target:=0;			
			PWM_Y2_Target:=REAL_TO_UINT(UINT_TO_REAL(PWM_JOYX_R_UP)/1000*(PAR_Y2_PosFull-PAR_Y2_NegFull)+PAR_Y2_NegFull);
		END_IF
		PWM_Y12_SET_Tatget:=REAL_TO_UINT(UINT_TO_REAL(PWM_JOYX_R_UP)/1000*(PAR_Valve1_PosFull-PAR_Valve1_NegFull)+PAR_Valve1_NegFull);
		PWM_Y61_SET_Tatget:=REAL_TO_UINT(UINT_TO_REAL(PWM_JOYX_R_UP)/1000*(PAR_Valve1_PosFull-PAR_Valve1_NegFull)+PAR_Valve1_NegFull);
		PWM_Y14_SET_Tatget:=REAL_TO_UINT(UINT_TO_REAL(PWM_JOYX_R_UP_b)/500*(PAR_Valve2_PosFull-PAR_Valve2_NegFull)+PAR_Valve2_NegFull);
		PWM_Y11_SET:=0;
		PWM_Y13_SET:=0;
		PWM_Y60_SET:=0;
		PWM_Y11_SET_Tatget:=0;
		PWM_Y13_SET_Tatget:=0;
		PWM_Y60_SET_Tatget:=0;
		IF(PWM_JOYX_R_UP>700)THEN
			PWM_Y41_SET:=PAR_Valve2_PosFull;//快速回油阀
		END_IF
		PWM_Y59_SET:=0;
		PWM_Y42_SET:=0;
	ELSIF PWM_JOYX_R_DOWN>10 THEN //动力头正转
			PWM_Y1_Target:=REAL_TO_UINT(UINT_TO_REAL(PWM_JOYX_R_DOWN)/1000*(PAR_Y1_PosFull-PAR_Y1_NegFull)+PAR_Y1_NegFull);			
			PWM_Y2_Target:=REAL_TO_UINT(UINT_TO_REAL(PWM_JOYX_R_DOWN_b)/500*(PAR_Y2_PosFull-PAR_Y2_NegFull)+PAR_Y2_NegFull);
		IF(DIH_SA18)THEN
			PWM_Y1_Target:=0;			
			PWM_Y2_Target:=REAL_TO_UINT(UINT_TO_REAL(PWM_JOYX_R_DOWN)/1000*(PAR_Y2_PosFull-PAR_Y2_NegFull)+PAR_Y2_NegFull);
		END_IF
			PWM_Y11_SET_Tatget:=REAL_TO_UINT(UINT_TO_REAL(PWM_JOYX_R_DOWN)/1000*(PAR_Valve1_PosFull-PAR_Valve1_NegFull)+PAR_Valve1_NegFull);
			PWM_Y60_SET_Tatget:=REAL_TO_UINT(UINT_TO_REAL(PWM_JOYX_R_DOWN)/1000*(PAR_Valve1_PosFull-PAR_Valve1_NegFull)+PAR_Valve1_NegFull);		
			PWM_Y13_SET_Tatget:=REAL_TO_UINT(UINT_TO_REAL(PWM_JOYX_R_DOWN_b)/500*(PAR_Valve2_PosFull-PAR_Valve2_NegFull)+PAR_Valve2_NegFull);
		IF(PWM_JOYX_R_DOWN>700)THEN
		PWM_Y59_SET:=PAR_Valve2_PosFull;//合流
		PWM_Y42_SET:=PAR_Valve2_PosFull;//快速回油阀
		END_IF
		PWM_Y41_SET:=0;
		PWM_Y12_SET:=0;
		PWM_Y14_SET:=0;
		PWM_Y61_SET:=0;	
		PWM_Y12_SET_Tatget:=0;
		PWM_Y14_SET_Tatget:=0;
		PWM_Y61_SET_Tatget:=0;
	END_IF
ELSIF (MainWinch_move) AND(PowerHead_move) AND( NOT DI_RHandle_SB6) THEN
	//主卷和动力头复合动作时 主泵2提供给动力头油
	IF PWM_JOYX_R_UP>10 THEN//动力头反转 
		IF(PWM_JOYY_L_DOWN>10) THEN//主卷上提
		PWM_JOY_P:=MAX(PWM_JOYY_L_DOWN,PWM_JOYX_R_UP);
		PWM_Y1_Target:=REAL_TO_UINT(UINT_TO_REAL(PWM_JOY_P)/1000*(PAR_Y2_PosFull-PAR_Y2_NegFull)+PAR_Y2_NegFull);
		PWM_Y12_SET_Tatget:=REAL_TO_UINT(UINT_TO_REAL(PWM_JOYX_R_UP)/1000*(PAR_Valve2_PosFull-400)*P_value+400);
		PWM_Y11_SET_Tatget:=0;
		PWM_Y14_SET_Tatget:=0;
		PWM_Y13_SET_Tatget:=0;
		PWM_Y60_SET_Tatget:=0;
		PWM_Y61_SET_Tatget:=0;
		PWM_Y41_SET:=PAR_Valve2_PosFull;
		PWM_Y42_SET:=0;
		PWM_Y59_SET:=0;
		ELSIF PWM_JOYY_L_UP>10 THEN//主卷下放
 		PWM_Y1_Target:=REAL_TO_UINT(UINT_TO_REAL(PWM_JOYX_R_UP)/1000*(PAR_Y2_PosFull-PAR_Y2_NegFull)+PAR_Y2_NegFull);
		PWM_Y12_SET_Tatget:=REAL_TO_UINT(UINT_TO_REAL(PWM_JOYX_R_UP)/1000*(PAR_Valve2_PosFull-PAR_Valve2_NegFull)+PAR_Valve2_NegFull);
		PWM_Y11_SET_Tatget:=0;
		PWM_Y14_SET_Tatget:=0;
		PWM_Y13_SET_Tatget:=0;
		PWM_Y60_SET_Tatget:=0;
		PWM_Y61_SET_Tatget:=0;
		PWM_Y41_SET:=PAR_Valve2_PosFull;
		PWM_Y59_SET:=0;	
		PWM_Y42_SET:=0;
		END_IF
		
		
	ELSIF PWM_JOYX_R_DOWN>10 THEN //动力头正转
		PWM_Y1_Target:=REAL_TO_UINT(UINT_TO_REAL(PWM_JOYX_R_DOWN)/1000*(PAR_Y2_PosFull-PAR_Y2_NegFull)+PAR_Y2_NegFull);
		PWM_Y11_SET_Tatget:=REAL_TO_UINT(UINT_TO_REAL(PWM_JOYX_R_DOWN)/1000*(PAR_Valve2_PosFull-PAR_Valve2_NegFull)+PAR_Valve2_NegFull);
		PWM_Y13_SET_Tatget:=0;
		PWM_Y12_SET_Tatget:=0;
		PWM_Y14_SET_Tatget:=0;
		PWM_Y60_SET_Tatget:=0;
		PWM_Y61_SET_Tatget:=0;
		PWM_Y41_SET:=0;
		PWM_Y42_SET:=PAR_Valve2_PosFull;
		PWM_Y59_SET:=0;	
	END_IF	
ELSE
		PWM_Y12_SET_Tatget:=0;
		PWM_Y14_SET_Tatget:=0;
		PWM_Y61_SET_Tatget:=0;
		PWM_Y11_SET_Tatget:=0;
		PWM_Y13_SET_Tatget:=0;
		PWM_Y60_SET_Tatget:=0;
		PWM_Y41_SET:=0;
		PWM_Y42_SET:=0;	
		PWM_Y59_SET:=0;	
END_IF


//判断抛土模式
Rtrig_DongLiTou1(clk:=(CANI_JOYX_R>3000));//反转判断
IF Rtrig_DongLiTou1.Q THEN
	Count_TIMES_Fanzhuan:=Count_TIMES_Fanzhuan + 1;
END_IF
Rtrig_DongLiTou2(clk:=(CANI_JOYX_R<2000));//正转判断
IF Rtrig_DongLiTou2.Q THEN
	Count_TIMES_Zhengzhuan:=Count_TIMES_Zhengzhuan + 1;
END_IF	
IF (Count_TIMES_Fanzhuan_LAST<>Count_TIMES_Fanzhuan) AND (Count_TIMES_Zhengzhuan_LAST<>Count_TIMES_Zhengzhuan) THEN
	Paotu_Modle:=TRUE;
END_IF
TIME_1000ms(IN:=NOT TIME_1000ms.Q,PT:=T#800MS);
IF (TIME_1000ms.Q) THEN
	Count_TIMES_Fanzhuan_LAST:=Count_TIMES_Fanzhuan;
	Count_TIMES_Zhengzhuan_LAST:=Count_TIMES_Zhengzhuan;
END_IF

IF(Count_TIMES_Fanzhuan_LAST=Count_TIMES_Fanzhuan) AND (Count_TIMES_Zhengzhuan_LAST=Count_TIMES_Zhengzhuan) THEN
	PaoTU_biaozhi:=TRUE;
ELSE
	PaoTU_biaozhi:=FALSE;	
END_IF
TIME_1000ms_TP(IN:=PaoTU_biaozhi,PT:=T#800MS);
IF TIME_1000ms_TP.Q OR MainWinch_move  THEN
	Paotu_Modle:=FALSE;
END_IF

IF(NOT CANI_WorkModeSwitch) THEN
	Paotu_Modle:=FALSE;
END_IF

IF Paotu_Modle THEN
	TIMEBASE_ratate:=T#20MS;
ELSE
	TIMEBASE_ratate:=T#100MS;
END_IF


(*动力头动作缓冲*)
//启动缓冲时间300ms，停止缓冲时间600ms
(*动力头动作缓冲*)
//启动缓冲时间300ms，停止缓冲时间600ms
RAMP1(
	IN:=WORD_TO_INT(PWM_Y11_SET_Tatget), 
	ASCEND:= R_RAMP_ratate, 
	DESCEND:= F_RAMP_ratate, 
	TIMEBASE:=TIMEBASE_ratate , 
	RESET:=FALSE , 
	OUT=>(PWM_Y11_SET_Tatget1));
IF(PWM_Y11_SET_Tatget1>=400) THEN
	Curve_input:=TO_UINT(PWM_Y11_SET_Tatget1 - 400);
	IF(Curve_input>900) THEN
		Curve_input:=900;
	END_IF
	curve1(input:=REAL_TO_UINT(UINT_TO_REAL(Curve_input)*72.8),Zero:=FALSE,Full:=FALSE,
		   PAR_Progression:=Curve_Par,OutputEnable:=TRUE);
	PWM_Y11_SET:=PAR_Valve1_NegFull + REAL_TO_UINT(UINT_TO_REAL(curve1.Output)/72.8);
ELSE
	PWM_Y11_SET:=0;
END_IF

RAMP2(
	IN:=WORD_TO_INT(PWM_Y12_SET_Tatget), 
	ASCEND:= R_RAMP_ratate, 
	DESCEND:= F_RAMP_ratate, 
	TIMEBASE:=TIMEBASE_ratate , 
	RESET:=FALSE , 
	OUT=>(PWM_Y12_SET_Tatget1));
IF(PWM_Y12_SET_Tatget1>=400) THEN
	Curve_input:=TO_UINT(PWM_Y12_SET_Tatget1 - 400);
	IF(Curve_input>900) THEN
		Curve_input:=900;
	END_IF
	curve2(input:=REAL_TO_UINT(UINT_TO_REAL(Curve_input)*72.8),Zero:=FALSE,Full:=FALSE,
		   PAR_Progression:=Curve_Par,OutputEnable:=TRUE);
	PWM_Y12_SET:=PAR_Valve1_NegFull + REAL_TO_UINT(UINT_TO_REAL(curve2.Output)/72.8);
ELSE
	PWM_Y12_SET:=0;
END_IF

RAMP3(
	IN:=WORD_TO_INT(PWM_Y13_SET_Tatget), 
	ASCEND:= R_RAMP_ratate, 
	DESCEND:= F_RAMP_ratate, 
	TIMEBASE:=TIMEBASE_ratate , 
	RESET:=FALSE , 
	OUT=>(PWM_Y13_SET_Tatget1));
IF(PWM_Y13_SET_Tatget1>=400) THEN
	Curve_input:=TO_UINT(PWM_Y13_SET_Tatget1 - 400);
	IF(Curve_input>900) THEN
		Curve_input:=900;
	END_IF
	curve3(input:=REAL_TO_UINT(UINT_TO_REAL(Curve_input)*72.8),Zero:=FALSE,Full:=FALSE,
		   PAR_Progression:=Curve_Par,OutputEnable:=TRUE);
	PWM_Y13_SET:=PAR_Valve1_NegFull + REAL_TO_UINT(UINT_TO_REAL(curve3.Output)/72.8);
ELSE
	PWM_Y13_SET:=0;
END_IF

RAMP4(
	IN:=WORD_TO_INT(PWM_Y14_SET_Tatget), 
	ASCEND:= R_RAMP_ratate, 
	DESCEND:= F_RAMP_ratate, 
	TIMEBASE:=TIMEBASE_ratate , 
	RESET:=FALSE , 
	OUT=>(PWM_Y14_SET_Tatget1));
IF(PWM_Y14_SET_Tatget1>=400) THEN
	Curve_input:=TO_UINT(PWM_Y14_SET_Tatget1 - 400);
	IF(Curve_input>900) THEN
		Curve_input:=900;
	END_IF
	curve4(input:=REAL_TO_UINT(UINT_TO_REAL(Curve_input)*72.8),Zero:=FALSE,Full:=FALSE,
		   PAR_Progression:=Curve_Par,OutputEnable:=TRUE);
	PWM_Y14_SET:=PAR_Valve1_NegFull + REAL_TO_UINT(UINT_TO_REAL(curve4.Output)/72.8);
ELSE
	PWM_Y14_SET:=0;
END_IF

RAMP5(
	IN:=WORD_TO_INT(PWM_Y60_SET_Tatget), 
	ASCEND:= R_RAMP_ratate, 
	DESCEND:= F_RAMP_ratate, 
	TIMEBASE:=TIMEBASE_ratate , 
	RESET:=FALSE , 
	OUT=>(PWM_Y60_SET_Tatget1));
IF(PWM_Y60_SET_Tatget1>=400) THEN
	Curve_input:=TO_UINT(PWM_Y60_SET_Tatget1 - 400);
	IF(Curve_input>900) THEN
		Curve_input:=900;
	END_IF
	curve5(input:=REAL_TO_UINT(UINT_TO_REAL(Curve_input)*72.8),Zero:=FALSE,Full:=FALSE,
		   PAR_Progression:=Curve_Par,OutputEnable:=TRUE);
	PWM_Y60_SET:=PAR_Valve1_NegFull + REAL_TO_UINT(UINT_TO_REAL(curve5.Output)/72.8);
ELSE
	PWM_Y60_SET:=0;
END_IF

RAMP6(
	IN:=WORD_TO_INT(PWM_Y61_SET_Tatget), 
	ASCEND:= R_RAMP_ratate, 
	DESCEND:= F_RAMP_ratate, 
	TIMEBASE:=TIMEBASE_ratate , 
	RESET:=FALSE , 
	OUT=>(PWM_Y61_SET_Tatget1));
IF(PWM_Y61_SET_Tatget1>=400) THEN
	Curve_input:=TO_UINT(PWM_Y61_SET_Tatget1 - 400);
	IF(Curve_input>900) THEN
		Curve_input:=900;
	END_IF
	curve6(input:=REAL_TO_UINT(UINT_TO_REAL(Curve_input)*72.8),Zero:=FALSE,Full:=FALSE,
		   PAR_Progression:=Curve_Par,OutputEnable:=TRUE);
	PWM_Y61_SET:=PAR_Valve1_NegFull + REAL_TO_UINT(UINT_TO_REAL(curve6.Output)/72.8);
ELSE
	PWM_Y61_SET:=0;
END_IF


IF(PWM_Y5_SET>1300)THEN
	PWM_Y5_SET :=1300;
END_IF
IF(PWM_Y6_SET>1300)THEN
	PWM_Y6_SET :=1300;
END_IF
IF(PWM_Y15_SET>1300)THEN
	PWM_Y15_SET :=1300;
END_IF
IF(PWM_Y16_SET>1300)THEN
	PWM_Y16_SET :=1300;
END_IF	
IF(PWM_Y11_SET>1300)THEN
	PWM_Y11_SET :=1300;
END_IF
IF(PWM_Y12_SET>1300)THEN
	PWM_Y12_SET :=1300;
END_IF
IF(PWM_Y13_SET>1300)THEN
	PWM_Y13_SET :=1300;
END_IF
IF(PWM_Y14_SET>1300)THEN
	PWM_Y14_SET :=1300;
END_IF
IF(PWM_Y60_SET>1300)THEN
	PWM_Y60_SET :=1300;
END_IF
IF(PWM_Y61_SET>1300)THEN
	PWM_Y61_SET :=1300;
END_IF


IF(PWM_Y11_SET<=300)THEN
	PWM_Y11_SET :=0;
END_IF
IF(PWM_Y12_SET<=300)THEN
	PWM_Y12_SET :=0;
END_IF
IF(PWM_Y13_SET<=300)THEN
	PWM_Y13_SET :=0;
END_IF
IF(PWM_Y14_SET<=300)THEN
	PWM_Y14_SET :=0;
END_IF
IF(PWM_Y60_SET<=300)THEN
	PWM_Y60_SET :=0;
END_IF
IF(PWM_Y61_SET<=300)THEN
	PWM_Y61_SET :=0;
END_IF


BiaoZHI_MainWinchUp:=FALSE;
IF(PWM_JOYY_L_UP<=500)THEN
	PWM_JOYY_L_UP_a:=PWM_JOYY_L_UP;
	PWM_JOYY_L_UP_b:=0;
ELSE
	PWM_JOYY_L_UP_a:=500;
	PWM_JOYY_L_UP_b:=PWM_JOYY_L_UP-500;
END_IF

IF(PWM_JOYY_L_DOWN<=500)THEN
	PWM_JOYY_L_DOWN_a:=PWM_JOYY_L_DOWN;
	PWM_JOYY_L_DOWN_b:=0;
ELSE
	PWM_JOYY_L_DOWN_a:=500;
	PWM_JOYY_L_DOWN_b:=PWM_JOYY_L_DOWN-500;
END_IF



(*单主卷动作*)
IF ( MainWinch_move) AND (NOT PowerHead_move) AND (NOT LeftMove_move) AND (NOT RightMove_move)THEN
	IF PWM_JOYY_L_UP>10   THEN//主卷下放
		PWM_Y1_Target:=REAL_TO_UINT(UINT_TO_REAL(PWM_JOYY_L_UP)/1000*(PAR_Y1_PosFull-PAR_Y1_NegFull)+PAR_Y1_NegFull);
		PWM_Y2_Target:=REAL_TO_UINT(UINT_TO_REAL(PWM_JOYY_L_UP)/1000*(PAR_Y2_PosFull-PAR_Y2_NegFull)+PAR_Y2_NegFull);
		BiaoZHI_MainWinchUp:=TRUE;
		PWM_Y8_SET_Target:=REAL_TO_UINT(UINT_TO_REAL(PWM_JOYY_L_UP)/1000*(PAR_Valve1_PosFull-PAR_Valve1_NegFull)+PAR_Valve1_NegFull);
		PWM_Y10_SET_Target:=REAL_TO_UINT(UINT_TO_REAL(PWM_JOYY_L_UP)/1000*(PAR_Valve2_PosFull-PAR_Valve2_NegFull)+PAR_Valve2_NegFull);
		PWM_Y7_SET_Target:=0;
		PWM_Y9_SET_Target:=0;
		IF(DIH_SA19)THEN
			PWM_Y10_SET_Target:=0;
			PWM_Y9_SET_Target:=0;
			PWM_Y2_Target:=0;	
		END_IF
	ELSIF PWM_JOYY_L_DOWN>10 THEN//主卷上提
		PWM_Y1_Target:=REAL_TO_UINT(UINT_TO_REAL(PWM_JOYY_L_DOWN)/1000*(PAR_Y1_PosFull-PAR_Y1_NegFull)+PAR_Y1_NegFull);
		PWM_Y2_Target:=REAL_TO_UINT(UINT_TO_REAL(PWM_JOYY_L_DOWN)/1000*(PAR_Y2_PosFull-PAR_Y2_NegFull)+PAR_Y2_NegFull);
		PWM_Y7_SET_Target:=REAL_TO_UINT(UINT_TO_REAL(PWM_JOYY_L_DOWN)/1000*(PAR_Valve1_PosFull-PAR_Valve2_NegFull)+PAR_Valve2_NegFull);
		PWM_Y9_SET_Target:=REAL_TO_UINT(UINT_TO_REAL(PWM_JOYY_L_DOWN)/1000*(PAR_Valve2_PosFull-PAR_Valve2_NegFull)+PAR_Valve2_NegFull);
		PWM_Y8_SET_Target:=0;
		PWM_Y10_SET_Target:=0;	
		IF(DIH_SA19)THEN
			PWM_Y10_SET_Target:=0;
			PWM_Y9_SET_Target:=0;
			PWM_Y2_Target:=0;	
		END_IF
	END_IF
ELSIF( MainWinch_move) AND (PowerHead_move) THEN
	//主卷和动力头复合动作时 主泵1提供给主卷油
	IF PWM_JOYY_L_UP>10 THEN//主卷下放
		IF(PWM_JOYX_R_DOWN>10) THEN //动力头正转
			PWM_JOY_P4:=MAX(PWM_JOYY_L_UP,PWM_JOYX_R_DOWN);
			PWM_Y2_Target:=REAL_TO_UINT(UINT_TO_REAL(PWM_JOYY_L_UP)/1000*(PAR_Y1_PosFull-PAR_Y1_NegFull)+PAR_Y1_NegFull);
			PWM_Y1_Target:=REAL_TO_UINT(UINT_TO_REAL(PWM_JOYY_L_UP)/1000*(PAR_Y1_PosFull-PAR_Y1_NegFull)+PAR_Y1_NegFull);
			PWM_Y10_SET_Target:=REAL_TO_UINT(UINT_TO_REAL(PWM_JOYY_L_UP)/1000*(PAR_Valve1_PosFull-PAR_Valve1_NegFull)+PAR_Valve1_NegFull);
			PWM_Y8_SET_Target:=REAL_TO_UINT(UINT_TO_REAL(1000-PWM_JOYX_R_DOWN)/1000*(PAR_Valve1_PosFull-PAR_Valve1_NegFull)+PAR_Valve1_NegFull);
			PWM_Y7_SET_Target:=0;
			PWM_Y9_SET_Target:=0;
		ELSIF PWM_JOYX_R_UP>10 THEN//动力头反转
			PWM_JOY_P3:=MAX(PWM_JOYY_L_UP,PWM_JOYX_R_UP);
			PWM_Y2_Target:=REAL_TO_UINT(UINT_TO_REAL(PWM_JOYY_L_UP)/1000*(PAR_Y1_PosFull-PAR_Y1_NegFull)+PAR_Y1_NegFull);
			PWM_Y1_Target:=REAL_TO_UINT(UINT_TO_REAL(PWM_JOYY_L_UP)/1000*(PAR_Y1_PosFull-PAR_Y1_NegFull)+PAR_Y1_NegFull);
			PWM_Y10_SET_Target:=REAL_TO_UINT(UINT_TO_REAL(PWM_JOYY_L_UP)/1000*(PAR_Valve1_PosFull-PAR_Valve1_NegFull)+PAR_Valve1_NegFull);
			PWM_Y8_SET_Target:=REAL_TO_UINT(UINT_TO_REAL(1000-PWM_JOYX_R_UP)/1000*(PAR_Valve1_PosFull-PAR_Valve1_NegFull)+PAR_Valve1_NegFull);
			PWM_Y7_SET_Target:=0;
			PWM_Y9_SET_Target:=0;
		END_IF	
	ELSIF PWM_JOYY_L_DOWN>10 THEN//主卷上提
		IF(PWM_JOYX_R_DOWN>10) THEN //动力头正转
			PWM_JOY_P2:=MAX(PWM_JOYY_L_DOWN,PWM_JOYX_R_DOWN);
			PWM_Y2_Target:=REAL_TO_UINT(UINT_TO_REAL(PWM_JOYY_L_DOWN)/1000*(PAR_Y1_PosFull-PAR_Y1_NegFull)+PAR_Y1_NegFull);
			PWM_Y1_Target:=REAL_TO_UINT(UINT_TO_REAL(PWM_JOYY_L_DOWN)/1000*(PAR_Y1_PosFull-PAR_Y1_NegFull)+PAR_Y1_NegFull);
			PWM_Y9_SET_Target:=REAL_TO_UINT(UINT_TO_REAL(PWM_JOYY_L_DOWN)/1000*(PAR_Valve1_PosFull-750)+750);
			PWM_Y7_SET_Target:=REAL_TO_UINT(UINT_TO_REAL(PWM_JOYY_L_DOWN)/1000*(PAR_Valve1_PosFull-750)+750);
			PWM_Y8_SET_Target:=0;
			PWM_Y10_SET_Target:=0;
		ELSIF PWM_JOYX_R_UP>10 THEN//动力头反转
			PWM_JOY_P1:=MAX(PWM_JOYY_L_DOWN,PWM_JOYX_R_UP);
			PWM_Y1_Target:=REAL_TO_UINT(UINT_TO_REAL(PWM_JOYY_L_DOWN)/1000*(PAR_Y1_PosFull-PAR_Y1_NegFull)+PAR_Y1_NegFull);
			PWM_Y2_Target:=REAL_TO_UINT(UINT_TO_REAL(PWM_JOYY_L_DOWN)/1000*(PAR_Y2_PosFull-PAR_Y2_NegFull)+PAR_Y2_NegFull);
			PWM_Y7_SET_Target:=REAL_TO_UINT(UINT_TO_REAL(PWM_JOYY_L_DOWN)/1000*(PAR_Valve1_PosFull-750)+750);
			PWM_Y9_SET_Target:=REAL_TO_UINT(UINT_TO_REAL(PWM_JOYY_L_DOWN)/1000*(PAR_Valve2_PosFull-750)+750);
			PWM_Y8_SET_Target:=0;
			PWM_Y10_SET_Target:=0;
		END_IF
	END_IF
ELSIF (MainWinch_move) AND (LeftMove_move OR RightMove_move) THEN
//主卷和行走复合动作 主泵1提供给主卷油
	IF PWM_JOYY_L_UP>10 THEN//主卷下放
		PWM_Y1_Target:=REAL_TO_UINT(UINT_TO_REAL(PWM_JOYY_L_UP)/1000*(PAR_Y1_PosFull-PAR_Y1_NegFull)+PAR_Y1_NegFull);
		PWM_Y10_SET_Target:=0;
		PWM_Y8_SET_Target:=PAR_Valve1_PosFull;
		PWM_Y7_SET_Target:=0;
		PWM_Y9_SET_Target:=0;
	ELSIF PWM_JOYY_L_DOWN>10 THEN//主卷上提
		PWM_Y1_Target:=REAL_TO_UINT(UINT_TO_REAL(PWM_JOYY_L_DOWN)/1000*(PAR_Y1_PosFull-PAR_Y1_NegFull)+PAR_Y1_NegFull);
		PWM_Y9_SET_Target:=0;
		PWM_Y7_SET_Target:=PAR_Valve1_PosFull;
		PWM_Y8_SET_Target:=0;
		PWM_Y10_SET_Target:=0;		
		PWM_Y19_SET:=0;
		IF(DI_LHandle_SB4)THEN
			PWM_Y20_SET:=600;
		ELSE
			PWM_Y20_SET:=0;
		END_IF
	END_IF
ELSE
		PWM_Y8_SET:=0;
		PWM_Y10_SET:=0;
		PWM_Y7_SET:=0;
		PWM_Y9_SET:=0;
		PWM_Y8_SET_Target:=0;
		PWM_Y10_SET_Target:=0;
		PWM_Y7_SET_Target:=0;
		PWM_Y9_SET_Target:=0;
END_IF
	
	
//主卷扬根据阀的开关调整斜坡值	
	IF(PWM_Y8_SET<1000  AND  PWM_Y8_SET>=900)THEN    //主卷下放斜坡值
			F_RAMP_mainwinch_down:=200;
	ELSIF(PWM_Y8_SET<900)THEN
			F_RAMP_mainwinch_down:=100;
	ELSE
			F_RAMP_mainwinch_down:=200;
	END_IF
		
	IF(PWM_Y7_SET<1000  AND  PWM_Y7_SET>=900)THEN  //主卷上提斜坡值
			F_RAMP_mainwinch_down:=300;
	ELSIF(PWM_Y7_SET<900  )THEN
			F_RAMP_mainwinch_down:=200;
	ELSE
			F_RAMP_mainwinch_down:=400;
	END_IF
		
RAMP7(
	IN:=WORD_TO_INT(PWM_Y7_SET_Target), 
	ASCEND:= R_RAMP_mainwinch, 
	DESCEND:= F_RAMP_mainwinch_up, 
	TIMEBASE:=TIMEBASE_mainwinch , 
	RESET:=FALSE , 
	OUT=>(PWM_Y7_SET_Target1));
IF(PWM_Y7_SET_Target1>=400) THEN
	Curve_input:=TO_UINT(PWM_Y7_SET_Target1 - 400);
	IF(Curve_input>900) THEN
		Curve_input:=900;
	END_IF
	curve7(input:=REAL_TO_UINT(UINT_TO_REAL(Curve_input)*72.8),Zero:=FALSE,Full:=FALSE,
		   PAR_Progression:=Curve_Par,OutputEnable:=TRUE);
	PWM_Y7_SET:=PAR_Valve1_NegFull + REAL_TO_UINT(UINT_TO_REAL(curve7.Output)/72.8);
ELSE
	PWM_Y7_SET:=0;
END_IF


RAMP8(
	IN:=WORD_TO_INT(PWM_Y8_SET_Target), 
	ASCEND:= R_RAMP_mainwinch, 
	DESCEND:= F_RAMP_mainwinch_down, 
	TIMEBASE:=TIMEBASE_mainwinch , 
	RESET:=FALSE , 
	OUT=>(PWM_Y8_SET_Target1));
IF(PWM_Y8_SET_Target1>=400) THEN
	Curve_input:=TO_UINT(PWM_Y8_SET_Target1 - 400);
	IF(Curve_input>900) THEN
		Curve_input:=900;
	END_IF
	curve8(input:=REAL_TO_UINT(UINT_TO_REAL(Curve_input)*72.8),Zero:=FALSE,Full:=FALSE,
		   PAR_Progression:=Curve_Par,OutputEnable:=TRUE);
	PWM_Y8_SET:=PAR_Valve1_NegFull + REAL_TO_UINT(UINT_TO_REAL(curve8.Output)/72.8);
ELSE
	PWM_Y8_SET:=0;
END_IF


RAMP9(
	IN:=WORD_TO_INT(PWM_Y9_SET_Target), 
	ASCEND:= R_RAMP_mainwinch, 
	DESCEND:= F_RAMP_mainwinch_up, 
	TIMEBASE:=TIMEBASE_mainwinch , 
	RESET:=FALSE , 
	OUT=>(PWM_Y9_SET_Target1));
IF(PWM_Y9_SET_Target1>=400) THEN
	Curve_input:=TO_UINT(PWM_Y9_SET_Target1 - 400);
	IF(Curve_input>900) THEN
		Curve_input:=900;
	END_IF
	curve9(input:=REAL_TO_UINT(UINT_TO_REAL(Curve_input)*72.8),Zero:=FALSE,Full:=FALSE,
		   PAR_Progression:=Curve_Par,OutputEnable:=TRUE);
	PWM_Y9_SET:=PAR_Valve1_NegFull + REAL_TO_UINT(UINT_TO_REAL(curve9.Output)/72.8);
ELSE
	PWM_Y9_SET:=0;
END_IF

RAMP10(
	IN:=WORD_TO_INT(PWM_Y10_SET_Target), 
	ASCEND:= R_RAMP_mainwinch, 
	DESCEND:= F_RAMP_mainwinch_down, 
	TIMEBASE:=TIMEBASE_mainwinch , 
	RESET:=FALSE , 
	OUT=>(PWM_Y10_SET_Target1));
IF(PWM_Y10_SET_Target1>=400) THEN
	Curve_input:=TO_UINT(PWM_Y10_SET_Target1 - 400);
	IF(Curve_input>900) THEN
		Curve_input:=900;
	END_IF
	curve10(input:=REAL_TO_UINT(UINT_TO_REAL(Curve_input)*72.8),Zero:=FALSE,Full:=FALSE,
		   PAR_Progression:=Curve_Par,OutputEnable:=TRUE);
	PWM_Y10_SET:=PAR_Valve1_NegFull + REAL_TO_UINT(UINT_TO_REAL(curve10.Output)/72.8);
ELSE
	PWM_Y10_SET:=0;
END_IF


IF(PWM_Y7_SET>1300)THEN
	PWM_Y7_SET :=1300;
END_IF
IF(PWM_Y8_SET>1300)THEN
	PWM_Y8_SET :=1300;
END_IF
IF(PWM_Y9_SET>1300)THEN
	PWM_Y9_SET :=1300;
END_IF
IF(PWM_Y10_SET>1300)THEN
	PWM_Y10_SET :=1300;
END_IF

IF(PWM_Y7_SET<=300)THEN
	PWM_Y7_SET :=0;
END_IF
IF(PWM_Y8_SET<=300)THEN
	PWM_Y8_SET :=0;
END_IF
IF(PWM_Y9_SET<=300)THEN
	PWM_Y9_SET :=0;
END_IF
IF(PWM_Y10_SET<=300)THEN
	PWM_Y10_SET :=0;
END_IF




(*主泵卸荷阀控制*)
		PWM_Y39_SET_Target:=MAX(PWM_Y8_SET_Target,PWM_Y7_SET_Target,PWM_Y12_SET_Tatget,PWM_Y11_SET_Tatget,PWM_Y3_SET,PWM_Y4_SET,PWM_Y15_SET_Target,PWM_Y16_SET_Target);
		PWM_Y40_SET_Target:=MAX(PWM_Y9_SET_Target,PWM_Y10_SET_Target,PWM_Y13_SET_Tatget,PWM_Y14_SET_Tatget,PWM_Y5_SET_Target,PWM_Y6_SET_Target,PWM_Y17_SET2,PWM_Y18_SET);
	(*卸荷动作缓冲*)
RAMP19(
	IN:=WORD_TO_INT(PWM_Y39_SET_Target), 
	ASCEND:= R_RAMP_xiehe, 
	DESCEND:= F_RAMP_xiehe, 
	TIMEBASE:=TIMEBASE_xiehe , 
	RESET:=FALSE , 
	OUT=>(PWM_Y39_SET_Target1));
IF(PWM_Y39_SET_Target1>=400) THEN
	Curve_input:=TO_UINT(PWM_Y39_SET_Target1 - 400);
	IF(Curve_input>900) THEN
		Curve_input:=900;
	END_IF
	curve19(input:=REAL_TO_UINT(UINT_TO_REAL(Curve_input)*72.8),Zero:=FALSE,Full:=FALSE,
		   PAR_Progression:=Curve_Par1,OutputEnable:=TRUE);
	PWM_Y39_SET:=PAR_Valve1_NegFull + REAL_TO_UINT(UINT_TO_REAL(curve19.Output)/72.8);
ELSE
	PWM_Y39_SET:=0;
END_IF


RAMP20(
	IN:=WORD_TO_INT(PWM_Y40_SET_Target), 
	ASCEND:= R_RAMP_xiehe, 
	DESCEND:= F_RAMP_xiehe, 
	TIMEBASE:=TIMEBASE_xiehe , 
	RESET:=FALSE , 
	OUT=>(PWM_Y40_SET_Target1));
IF(PWM_Y40_SET_Target1>=400) THEN
	Curve_input:=TO_UINT(PWM_Y40_SET_Target1 - 400);
	IF(Curve_input>900) THEN
		Curve_input:=900;
	END_IF
	curve20(input:=REAL_TO_UINT(UINT_TO_REAL(Curve_input)*72.8),Zero:=FALSE,Full:=FALSE,
		   PAR_Progression:=Curve_Par1,OutputEnable:=TRUE);
	PWM_Y40_SET:=PAR_Valve1_NegFull + REAL_TO_UINT(UINT_TO_REAL(curve20.Output)/72.8);
ELSE
	PWM_Y40_SET:=0;
END_IF

	//在行走时一个泵供油时,需要关闭另外一个 泵的起压阀
	IF PWM_Y37_SET>500 AND (NOT MainWinch_move) THEN
		PWM_Y39_SET:=0;
	END_IF
	
IF(PWM_Y39_SET>1300)THEN
	PWM_Y39_SET :=1300;
END_IF
IF(PWM_Y40_SET>1300)THEN
	PWM_Y40_SET :=1300;
END_IF

IF(PWM_Y39_SET<=300)THEN
	PWM_Y39_SET :=0;
END_IF
IF(PWM_Y40_SET<=300)THEN
	PWM_Y40_SET :=0;
END_IF

(*副卷扬动作*)
IF(ViceWinch_move)THEN
	IF PWM_JOYY_R_UP>10 THEN//副卷下放
		PWM_Y4_SET:=REAL_TO_UINT(UINT_TO_REAL(PWM_JOYY_R_UP)/1000*(1200-500)+500);
		PWM_Y3_SET:=0;
		IF(NOT MainWinch_move) OR (NOT PowerHead_move) THEN
			PWM_Y1_Target:=REAL_TO_UINT(UINT_TO_REAL(PWM_JOYY_R_UP)/1000*(PAR_KP-PAR_Y1_NegFull)+PAR_Y1_NegFull);
		END_IF
		
	ELSIF PWM_JOYY_R_DOWN>10 THEN//副卷上提
		PWM_Y3_SET:=REAL_TO_UINT(UINT_TO_REAL(PWM_JOYY_R_DOWN)/1000*(1200-500)+500);
		PWM_Y4_SET:=0;
		IF(NOT MainWinch_move) OR (NOT PowerHead_move) THEN
			PWM_Y1_Target:=REAL_TO_UINT(UINT_TO_REAL(PWM_JOYY_R_DOWN)/1000*(PAR_KP-PAR_Y1_NegFull)+PAR_Y1_NegFull);
		END_IF		
	END_IF
ELSE
	PWM_Y3_SET:=0;
	PWM_Y4_SET:=0;
END_IF

(*回转动作*)
//回转限制
IF  (CANO_DEPTH>980 AND  CANI_WorkModeSwitch) THEN
		Rotation_move:=FALSE;
END_IF
	
IF NOT DI_LHandle_SB7 THEN(*自动回转*) 
	IF  Rotation_move  OR DI_LHandle_SB2  THEN
		DOH_Y50_1 := TRUE;
		IF PWM_JOYX_L_UP>10 THEN// 右回转
			PWM_Y22_SET:=REAL_TO_UINT(UINT_TO_REAL(PWM_JOYX_L_UP)/1000*(PAR_ValveC_NegFull-PAR_Valve3_NegFull)+PAR_Valve3_NegFull);
			PWM_Y21_SET:=0;
		ELSIF PWM_JOYX_L_DOWN>10 THEN//左回转
			PWM_Y21_SET:=REAL_TO_UINT(UINT_TO_REAL(PWM_JOYX_L_DOWN)/1000*(PAR_ValveC_NegFull-PAR_Valve3_NegFull)+PAR_Valve3_NegFull);
			PWM_Y22_SET:=0;
		END_IF
	ELSE
		DOH_Y50_1:= FALSE;
		PWM_Y21_SET:=0;
		PWM_Y22_SET:=0;
	END_IF
ELSE
	DOH_Y50_1 := TRUE;
	IF(AUTO_ROTATION_VALVE>=0) THEN
		PWM_Y21_SET:=REAL_TO_UINT(INT_TO_REAL(ABS(AUTO_ROTATION_VALVE))*0.13);
	ELSE
		PWM_Y22_SET:=REAL_TO_UINT(INT_TO_REAL(ABS(AUTO_ROTATION_VALVE))*0.13);		
	END_IF
END_IF

//回转时警示灯响并且监控显示后界面
IF Rotation_move  OR DOH_Y50 THEN
	DOH_70:=TRUE;
	DOH_73:=TRUE;
	DOH_JK2:=TRUE;
ELSE
	DOH_70:=FALSE;
	DOH_73:=FALSE;
	DOH_JK2:=FALSE;
END_IF

//制动阀延时锁车
Rotation_late(IN:=DOH_Y50_1,PT:=T#2S);
IF  DOH_Y50_1 THEN
	DOH_Y50:=TRUE;
ELSE
	DOH_Y50:=Rotation_late.Q;
END_IF

(*加压动作*)
IF JiaYa_move THEN
	IF PWM_JOYY_R_UP>10 THEN//加压下
		PWM_Y23_SET_Taget:=REAL_TO_UINT(UINT_TO_REAL(PWM_JOYY_R_UP)/1000*(800-PAR_Valve3_NegFull)+PAR_Valve3_NegFull);
		PWM_Y24_SET_Taget:=0;
		
		IF(CANI_JiaYaFastSwitch OR DI_RHandle_SB7)THEN //加压快
			PWM_Y2_Target:=REAL_TO_UINT(UINT_TO_REAL(PWM_JOYY_R_UP)/1000*(500-300)+300);
			PWM_Y17_SET:=0;
			PWM_Y17_SET2:=0;
			PWM_Y18_SET_Taget:=1300;
		ELSE
			PWM_Y18_SET_Taget:=0;
		END_IF
		
	ELSIF PWM_JOYY_R_DOWN>10 THEN//加压上
		PWM_Y24_SET_Taget:=REAL_TO_UINT(UINT_TO_REAL(PWM_JOYY_R_DOWN)/1000*(800-PAR_Valve3_NegFull)+PAR_Valve3_NegFull);
		PWM_Y23_SET_Taget:=0;
		
		IF(CANI_JiaYaFastSwitch OR DI_RHandle_SB7)THEN //加压快
			PWM_Y2_Target:=REAL_TO_UINT(UINT_TO_REAL(PWM_JOYY_R_DOWN)/1000*(500-300)+300);
			PWM_Y17_SET:=800;
			PWM_Y17_SET2:=1300;
			PWM_Y18_SET:=0;
		ELSE
			PWM_Y18_SET:=0;
		END_IF
	END_IF
ELSE
	PWM_Y23_SET_Taget:=0;
	PWM_Y24_SET_Taget:=0;
	PWM_Y17_SET:=0;
	PWM_Y18_SET:=0;
	PWM_Y17_SET2:=0;
END_IF

RAMP22(
	IN:=WORD_TO_INT(PWM_Y23_SET_Taget), 
	ASCEND:= ASCEND_value, 
	DESCEND:= 5000, 
	TIMEBASE:=T#1000MS , 
	RESET:=FALSE , 
	OUT=>(PWM_Y23_SET_Taget1));
IF(PWM_Y23_SET_Taget1<310)THEN
		ASCEND_value:=6000;
ELSIF(PWM_Y23_SET_Taget1>=310 AND PWM_Y23_SET_Taget1<450)THEN
		ASCEND_value:=100;
ELSE
		ASCEND_value:=300;
END_IF
IF(PWM_Y23_SET_Taget1>=300) THEN
	Curve_input:=TO_UINT(PWM_Y23_SET_Taget1 - 300);
	IF(Curve_input>500) THEN
		Curve_input:=500;
	END_IF
	PWM_Y23_SET:=300 + Curve_input;
ELSE
	PWM_Y23_SET:=0;
END_IF

RAMP24(
	IN:=WORD_TO_INT(PWM_Y24_SET_Taget), 
	ASCEND:= 500, 
	DESCEND:= 500, //500-6000
	TIMEBASE:=T#300MS , 
	RESET:=FALSE , 
	OUT=>((PWM_Y24_SET)));
(*IF(PWM_Y24_SET_Taget1>=300) THEN
	Curve_input:=TO_UINT(PWM_Y24_SET_Taget1 - 300);
	IF(Curve_input>500) THEN
		Curve_input:=500;
	END_IF
	PWM_Y24_SET:=300 + Curve_input;
ELSE
	PWM_Y24_SET:=0;
END_IF*)



RAMP23(
	IN:=WORD_TO_INT(PWM_Y18_SET_Taget), 
	ASCEND:= ASCEND_value2, 
	DESCEND:= 5000, 
	TIMEBASE:=T#1000MS , 
	RESET:=FALSE , 
	OUT=>(PWM_Y18_SET_Taget1));
IF(PWM_Y18_SET_Taget1<610)THEN
		ASCEND_value2:=6000;
ELSE
	ASCEND_value2:=150;
END_IF	

IF(PWM_Y18_SET_Taget1>=600) THEN
	Curve_input:=TO_UINT(PWM_Y18_SET_Taget1 - 600);
	IF(Curve_input>700) THEN
		Curve_input:=700;
	END_IF
	PWM_Y18_SET:=600 + Curve_input;
ELSE
	PWM_Y18_SET:=0;
END_IF

(*PWM_Y23_SET:=PWM_Y23_SET_Taget;*)
IF JiaYa_move THEN
	IF PWM_JOYY_R_DOWN>10 THEN
		PWM_Y23_SET_Taget:=0;
		PWM_Y23_SET_Taget1:=0;
		PWM_Y23_SET:=0;
		PWM_Y18_SET_Taget1:=0;
		PWM_Y18_SET_Taget:=0;
		PWM_Y18_SET:=0;
	END_IF
END_IF

//加压限压
IF(CANI_DongLiTouPressLimitSwitch)THEN
	PWM_Y63_SET:=PAR_ValveD_PosFull;
ELSE
	PWM_Y63_SET:=0;
END_IF
		
(*平举动作*)
IF  BianFu_move THEN
	IF PWM_JOYY_R_UP>10 THEN//变幅下
		PWM_Y25_SET:=REAL_TO_UINT(UINT_TO_REAL(PWM_JOYY_R_UP)/1000*(PAR_Valve3_PosFull-PAR_Valve3_NegFull)+PAR_Valve3_NegFull);
		PWM_Y26_SET:=0;
	ELSIF PWM_JOYY_R_DOWN>10 THEN//变幅上
		PWM_Y26_SET:=REAL_TO_UINT(UINT_TO_REAL(PWM_JOYY_R_DOWN)/1000*(PAR_Valve3_PosFull-PAR_Valve3_NegFull)+PAR_Valve3_NegFull);
		PWM_Y25_SET:=0;
	END_IF
ELSE
	PWM_Y25_SET:=0;
	PWM_Y26_SET:=0;
END_IF

(*张紧等切换油缸动作*)
IF  LvZhang_move THEN
	IF(NOT CANI_LvDaiShenSuoSwitch)THEN
		IF PWM_JOYX_R_UP>10 THEN
			PWM_Y31_SET:=REAL_TO_UINT(UINT_TO_REAL(PWM_JOYX_R_UP)/1000*(PAR_Valve3_PosFull-PAR_Valve3_NegFull)+PAR_Valve3_NegFull);
			PWM_Y32_SET:=0;
			PWM_Y19_SET:=0;
			PWM_Y20_SET:=0;
		ELSIF PWM_JOYX_R_DOWN>10 THEN
			PWM_Y32_SET:=REAL_TO_UINT(UINT_TO_REAL(PWM_JOYX_R_DOWN)/1000*(PAR_Valve3_PosFull-PAR_Valve3_NegFull)+PAR_Valve3_NegFull);
			PWM_Y31_SET:=0;
			PWM_Y19_SET:=0;
			PWM_Y20_SET:=0;
		ELSE
			PWM_Y31_SET:=0;
			PWM_Y32_SET:=0;
			PWM_Y19_SET:=0;
			PWM_Y20_SET:=0;
		END_IF
	ELSE
		IF PWM_JOYX_R_UP>10 THEN
			PWM_Y19_SET:=REAL_TO_UINT(UINT_TO_REAL(PWM_JOYX_R_UP)/1000*(PAR_Valve3_PosFull-PAR_Valve3_NegFull)+PAR_Valve3_NegFull);
			PWM_Y20_SET:=0;
			PWM_Y31_SET:=0;
			PWM_Y32_SET:=0;
		ELSIF PWM_JOYX_R_DOWN>10 THEN
			PWM_Y20_SET:=REAL_TO_UINT(UINT_TO_REAL(PWM_JOYX_R_DOWN)/1000*(PAR_Valve3_PosFull-PAR_Valve3_NegFull)+PAR_Valve3_NegFull);
			PWM_Y19_SET:=0;
			PWM_Y31_SET:=0;
			PWM_Y32_SET:=0;
		ELSE
			PWM_Y31_SET:=0;
			PWM_Y32_SET:=0;
			PWM_Y19_SET:=0;
			PWM_Y20_SET:=0;
		END_IF
	END_IF
ELSE
	PWM_Y31_SET:=0;
	PWM_Y32_SET:=0;
	PWM_Y19_SET:=0;
	PWM_Y20_SET:=0;
END_IF


IF(CANI_ETouYouGangSwitch) THEN//支腿/鹅头油缸切换
	DOH_Y52:=TRUE;
ELSE
	DOH_Y52:=FALSE;
END_IF

//主卷动作及浮动时开锁
IF  MainWinch_move OR DOH_Y55 THEN
	DOH_Y53 := TRUE;
	DOH_Y64:=TRUE;
	GVL_SaveEngine.Y74:=TRUE;
ELSE
	DOH_Y53 := FALSE;	
	DOH_Y64:=FALSE;
	GVL_SaveEngine.Y74:=FALSE;
END_IF

(*主泵功率控制20230706*)
//区分发动机转速
MainPump_Pressure_Taget1450:=PAR_NegFull_x;
MainPump_Pressure_Taget1600:=PAR_PosFull_x;
MainPump_Pressure_Taget1750:=PAR_Zero_x;

IF EngineSpeedTarget<=1080 THEN SPEED_CASE:=1;
ELSIF EngineSpeedTarget>1080 AND EngineSpeedTarget<=1300 THEN SPEED_CASE:=2;
ELSIF EngineSpeedTarget>1300 AND EngineSpeedTarget<=1520 THEN SPEED_CASE:=3;
ELSIF EngineSpeedTarget>1520 AND EngineSpeedTarget<=1680 THEN SPEED_CASE:=4;
ELSIF EngineSpeedTarget>1680 AND EngineSpeedTarget<=1820 THEN SPEED_CASE:=5;
ELSIF EngineSpeedTarget>1820 THEN SPEED_CASE:=6;;END_IF
//不同转速下的发动机最大功率
CASE SPEED_CASE OF
1:  Enginer_Power:=135;
2:  Enginer_Power:=174;
3:  Enginer_Power:=200;
4:  Enginer_Power:=230;
5:  Enginer_Power:=250;
6:  Enginer_Power:=261;
END_CASE
//不同转速下的压力值
IF(CANO_Fubeng_Press>100)THEN
	CASE SPEED_CASE OF
		1:MainPump_Pressure_Taget:=MainPump_Pressure_Taget1000-HELIU_Press_Target1000;
		2:MainPump_Pressure_Taget:=MainPump_Pressure_Taget1200-HELIU_Press_Target1200;
		3:MainPump_Pressure_Taget:=MainPump_Pressure_Taget1450-HELIU_Press_Target1400;
		4:MainPump_Pressure_Taget:=MainPump_Pressure_Taget1600-HELIU_Press_Target1600;
		5:MainPump_Pressure_Taget:=MainPump_Pressure_Taget1750-HELIU_Press_Target1800;
		6:MainPump_Pressure_Taget:=MainPump_Pressure_Taget1900-HELIU_Press_Target1900;
	END_CASE
ELSE
	CASE SPEED_CASE OF
		1:MainPump_Pressure_Taget:=MainPump_Pressure_Taget1000;
		2:MainPump_Pressure_Taget:=MainPump_Pressure_Taget1200;
		3:MainPump_Pressure_Taget:=MainPump_Pressure_Taget1450;
		4:MainPump_Pressure_Taget:=MainPump_Pressure_Taget1600;
		5:MainPump_Pressure_Taget:=MainPump_Pressure_Taget1750;
		6:MainPump_Pressure_Taget:=MainPump_Pressure_Taget1900;
	END_CASE		
END_IF
IF( CANI_ECOSwitch) THEN
	CASE SPEED_CASE OF
		1:MainPump_Pressure_Taget:=MainPump_Pressure_Taget1000-ECO_Press_Target1000;
		2:MainPump_Pressure_Taget:=MainPump_Pressure_Taget1200-ECO_Press_Target1200;
		3:MainPump_Pressure_Taget:=MainPump_Pressure_Taget1450-ECO_Press_Target1400;
		4:MainPump_Pressure_Taget:=MainPump_Pressure_Taget1600-ECO_Press_Target1600;
		5:MainPump_Pressure_Taget:=MainPump_Pressure_Taget1750-ECO_Press_Target1800;
		6:MainPump_Pressure_Taget:=MainPump_Pressure_Taget1900-ECO_Press_Target1900;
	END_CASE
END_IF
MainPump_Pressure:=CANO_MainPUMP_Press1+CANO_MainPUMP_Press2;
//消除滤波
MainPump_Pressure_Subtract:= UINT_TO_INT(MainPump_Pressure-MainPump_Pressure_last1);

TIME_200ms(IN:=NOT TIME_200ms.Q,PT:=T#400MS);

IF(TIME_200ms.Q)THEN
	CANI_JOYX_R_last:=CANI_JOYX_R;
END_IF
Sub_Joyx_r:=UINT_TO_INT(CANI_JOYX_R_last) - UINT_TO_INT(CANI_JOYX_R);
IF(Sub_Joyx_r<-1200 OR Sub_Joyx_r>1200) THEN
	Joyx_change_bool:=TRUE;
	
END_IF

IF(CANI_JOYX_R=2500)THEN
	tempbool:=TRUE;
ELSE
	tempbool:=FALSE;
END_IF

TIME_1000_1ms(in:=tempbool,PT:=T#500MS);
IF(TIME_1000_1ms.Q)THEN
	JOY_PAOTU:=FALSE;
END_IF

TIME_400ms(IN:=Joyx_change_bool,PT:=T#10MS);
IF(TIME_400ms.Q) THEN
	Joyx_change_bool:=FALSE;
END_IF



//大范围波动
IF MainPump_Pressure_Subtract>270 OR MainPump_Pressure_Subtract<-270 THEN
	Subtract:=TRUE;
ELSE
	Subtract:=FALSE;	
END_IF
	TIME_LvBo4(IN:=Subtract,PT:=T#10MS);
	
IF(TIME_LvBo4.Q) AND (CANO_MainPUMP_Press1>210) THEN 
		MainPump_Pressure_ChangeBool1:=TRUE;
END_IF
	TIME_LvBo1(IN:=MainPump_Pressure_ChangeBool1,PT:=T#2S);
IF(TIME_LvBo1.Q) THEN
	MainPump_Pressure_ChangeBool1 :=FALSE;
END_IF

IF(MainPump_Pressure_ChangeBool1) AND (MainPump_Pressure>MainPump_Pressure_last1) THEN 
	MainPump_Pressure_last1:=MainPump_Pressure;
END_IF

//小范围波动
t_powertime:=TO_TIME(PAR_DeadBand_x);
IF (NOT MainPump_Pressure_ChangeBool1) THEN
	IF(MainPump_Pressure_Subtract>40 OR MainPump_Pressure_Subtract<-40)THEN 
		MainPump_Pressure_ChangeBool:=TRUE;
	ELSE
		MainPump_Pressure_ChangeBool:=FALSE;
	END_IF

	TIME_LvBo2(IN:=MainPump_Pressure_ChangeBool,PT:=t_powertime);
	IF(TIME_LvBo2.Q )THEN
		MainPump_Pressure_last1:=MainPump_Pressure;
	END_IF	
END_IF


IF PowerHead_move AND NOT(MainWinch_move) THEN
		JianGE2:=0.005;
ELSE
	IF(EngineSpeedTarget>1000 AND EngineSpeedTarget<1300)THEN
		JianGE2:=0.005;
	ELSE
		JianGE2:=0.005;
	END_IF
END_IF
	
IF MainPump_Pressure_last1>MainPump_Pressure_Taget THEN
	Pressure_Coe_Taget:=UINT_TO_REAL(MainPump_Pressure_Taget)/UINT_TO_REAL(MainPump_Pressure_last1);(*压力系数*)
ELSE
	Pressure_Coe_Taget:=1;
END_IF
Pressure_Coe := Pressure_Coe_Taget;


IF MainPump_Pressure_last1>MainPump_Pressure_Taget  THEN
	IF(PWM_Y1_Target>=PAR_Y1_1_NegFull)THEN
		PWM_Y1_Target_OutPut:=REAL_TO_UINT(UINT_TO_REAL(PWM_Y1_Target-PAR_Y1_1_NegFull)*Pressure_Coe+PAR_Y1_1_NegFull);
	END_IF
	IF(PWM_Y2_Target>=PAR_Y1_1_NegFull)THEN
		PWM_Y2_Target_OutPut:=REAL_TO_UINT(UINT_TO_REAL(PWM_Y2_Target-PAR_Y1_1_NegFull)*Pressure_Coe+PAR_Y1_1_NegFull);
	END_IF
ELSE
	PWM_Y1_Target_OutPut:=PWM_Y1_Target;
	PWM_Y2_Target_OutPut:=PWM_Y2_Target;
END_IF

IF(EngineSpeedTarget>CANO_SPEED AND CANO_SPEED>400)THEN
	EngineSpeedSub:=EngineSpeedTarget - CANO_SPEED;
ELSE
	EngineSpeedSub:=0;
END_IF

IF(PWM_Y1_Target_OutPut<300)THEN PWM_Y1_Target_OutPut:=300;END_IF	
IF(PWM_Y2_Target_OutPut<300)THEN PWM_Y2_Target_OutPut:=300;END_IF

RAMP15_IN:=PWM_Y1_Target_OutPut;
RAMP16_IN:=PWM_Y2_Target_OutPut;


IF MainWinch_move  OR  LeftMove_move OR RightMove_move THEN  
	TIMEBASE_pump:=T#1000MS;
	TIMEBASE_xiehe:=T#500MS;
ELSE
	TIMEBASE_pump:=T#600MS;
	TIMEBASE_xiehe:=T#300MS;
END_IF
t_PowerHead_move(IN:= MainWinch_move,PT:=T#4S);
IF t_PowerHead_move.Q THEN
	F_RAMP_pump:=x_t_PowerHead_move;
	R_RAMP_pump:=x2_t_PowerHead_move;
ELSE
       CASE SPEED_CASE OF
                1:F_RAMP_pump:=1500; R_RAMP_pump:=100;                  
                2: 		IF MainWinch_move AND (JiaYa_move OR CANO_JiayaPressure>80)  THEN    //3泵同时起压时，降低主泵的加载速度，避免掉速熄火
                                F_RAMP_pump:=1500; R_RAMP_pump:=100;
                        ELSE
                                F_RAMP_pump:=1500; R_RAMP_pump:=100;//从200降
                                IF  PWM_JOYY_L_UP>10 THEN
                                 F_RAMP_pump:=1500; R_RAMP_pump:=200;
                                END_IF
                        END_IF            
                3:
                        IF MainWinch_move AND (JiaYa_move OR CANO_JiayaPressure>80)  THEN    //3泵同时起压时，降低主泵的加载速度，避免掉速熄火
                                F_RAMP_pump:=1500; R_RAMP_pump:=150;
                        ELSE
                                F_RAMP_pump:=1500; R_RAMP_pump:=TO_INT(PAR_NegFull_y);
                                IF  PWM_JOYY_L_UP>10 THEN
                                 F_RAMP_pump:=1500; R_RAMP_pump:=300;
                                END_IF
                        END_IF                
                4:
                        IF MainWinch_move AND (JiaYa_move OR CANO_JiayaPressure>80)  THEN
                                F_RAMP_pump:=1500; R_RAMP_pump:=150;
                        ELSE
                                F_RAMP_pump:=1500; R_RAMP_pump:=TO_INT(PAR_PosFull_y);//从200降
                                IF  PWM_JOYY_L_UP>10 THEN
                                 F_RAMP_pump:=1500; R_RAMP_pump:=300;
                                END_IF
                        END_IF                                
                5:
                        IF MainWinch_move AND (JiaYa_move OR CANO_JiayaPressure>80)  THEN
                                F_RAMP_pump:=1500; R_RAMP_pump:=200;
                        ELSE
                                F_RAMP_pump:=1500; R_RAMP_pump:=TO_INT(PAR_Zero_y);
                                IF  PWM_JOYY_L_UP>10 THEN
                                 F_RAMP_pump:=1500; R_RAMP_pump:=300;
                                END_IF
                        END_IF                        
                6:		IF MainWinch_move AND (JiaYa_move OR CANO_JiayaPressure>80)  THEN
                                F_RAMP_pump:=1500; R_RAMP_pump:=200;
                        ELSE
                                F_RAMP_pump:=1500; R_RAMP_pump:=200;
                                IF  PWM_JOYY_L_UP>10 THEN
                                 F_RAMP_pump:=1500; R_RAMP_pump:=300;
                                END_IF
                        END_IF               
         END_CASE	
END_IF

RAMP15(
	IN:=UINT_TO_INT(RAMP15_IN), 
	ASCEND:= R_RAMP_pump, 
	DESCEND:= F_RAMP_pump, 
	TIMEBASE:=TIMEBASE_pump , 
	RESET:=FALSE , 
	OUT=>(PWM_Y1_SET));
	
RAMP16(
	IN:=UINT_TO_INT(RAMP16_IN), 
	ASCEND:= R_RAMP_pump, 
	DESCEND:= F_RAMP_pump, 
	TIMEBASE:=TIMEBASE_pump , 
	RESET:=FALSE , 
	OUT=>(PWM_Y2_SET));

